C07311=1218.694,48.902,-44.910,-179.073,5.517,148.688
C07312=1218.690,49.151,-44.926,-179.071,5.518,148.687
C07313=1218.684,49.401,-44.942,-179.068,5.518,148.687
C07314=1218.680,49.650,-44.959,-179.065,5.519,148.686
C07315=1218.675,49.900,-44.975,-179.063,5.519,148.685
C07316=1218.670,50.149,-44.991,-179.060,5.520,148.685
C07317=1218.666,50.398,-45.007,-179.058,5.521,148.684
C07318=1218.660,50.648,-45.024,-179.055,5.521,148.684
C07319=1218.655,50.897,-45.041,-179.053,5.522,148.683
C07320=1218.650,51.146,-45.057,-179.050,5.522,148.682
C07321=1218.645,51.396,-45.073,-179.047,5.523,148.682
C07322=1218.641,51.645,-45.090,-179.045,5.524,148.681
C07323=1218.635,51.895,-45.107,-179.043,5.524,148.680
C07324=1218.630,52.145,-45.123,-179.040,5.525,148.680
C07325=1218.625,52.393,-45.139,-179.037,5.526,148.679
C07326=1218.621,52.643,-45.156,-179.035,5.526,148.678
C07327=1218.616,52.892,-45.172,-179.032,5.527,148.678
C07328=1218.611,53.141,-45.189,-179.030,5.528,148.677
C07329=1218.606,53.392,-45.205,-179.027,5.528,148.677
C07330=1218.601,53.641,-45.222,-179.025,5.529,148.676
C07331=1218.596,53.890,-45.238,-179.022,5.529,148.675
C07332=1218.591,54.140,-45.256,-179.019,5.530,148.675
C07333=1218.586,54.388,-45.272,-179.017,5.531,148.674
C07334=1218.581,54.638,-45.289,-179.015,5.531,148.674
C07335=1218.577,54.888,-45.305,-179.012,5.532,148.673
C07336=1218.571,55.156,-45.323,-179.009,5.532,148.672
C07337=1218.566,55.425,-45.341,-179.007,5.533,148.672
C07338=1218.561,55.693,-45.359,-179.004,5.534,148.671
C07339=1218.555,55.962,-45.377,-179.001,5.534,148.670
C07340=1218.550,56.211,-45.393,-178.999,5.535,148.670
C07341=1218.545,56.460,-45.410,-178.996,5.535,148.669
C07342=1218.540,56.710,-45.427,-178.993,5.536,148.668
C07343=1218.535,56.959,-45.443,-178.991,5.538,148.668
C07344=1218.531,57.208,-45.460,-178.988,5.538,148.667
C07345=1218.525,57.458,-45.477,-178.985,5.539,148.666
C07346=1218.520,57.707,-45.493,-178.983,5.539,148.666
C07347=1218.516,57.956,-45.510,-178.980,5.540,148.665
C07348=1218.511,58.206,-45.527,-178.978,5.541,148.665
C07349=1218.506,58.455,-45.544,-178.975,5.541,148.664
C07350=1218.501,58.705,-45.560,-178.973,5.542,148.663
C07351=1218.496,58.954,-45.578,-178.970,5.542,148.663
C07352=1218.491,59.204,-45.594,-178.967,5.543,148.662
C07353=1218.486,59.453,-45.611,-178.965,5.544,148.662
C07354=1218.481,59.702,-45.628,-178.963,5.544,148.661
C07355=1218.477,59.952,-45.644,-178.960,5.545,148.660
C07356=1218.471,60.201,-45.661,-178.957,5.546,148.660
C07357=1218.466,60.450,-45.678,-178.955,5.546,148.659
C07358=1218.462,60.700,-45.695,-178.953,5.547,148.659
C07359=1218.457,60.950,-45.712,-178.950,5.548,148.658
C07360=1218.452,61.199,-45.728,-178.947,5.548,148.657
C07361=1218.447,61.448,-45.746,-178.945,5.549,148.657
C07362=1218.442,61.697,-45.763,-178.943,5.550,148.656
C07363=1218.437,61.947,-45.780,-178.940,5.550,148.655
C07364=1218.432,62.196,-45.797,-178.937,5.551,148.655
C07365=1218.427,62.445,-45.813,-178.935,5.551,148.654
C07366=1218.422,62.695,-45.830,-178.932,5.552,148.653
C07367=1218.418,62.945,-45.847,-178.930,5.553,148.653
C07368=1218.412,63.194,-45.864,-178.927,5.553,148.652
C07369=1218.408,63.442,-45.881,-178.924,5.555,148.652
C07370=1218.402,63.692,-45.899,-178.921,5.555,148.651
C07371=1218.398,63.942,-45.915,-178.919,5.556,148.650
C07372=1218.393,64.192,-45.933,-178.917,5.557,148.650
C07373=1218.388,64.440,-45.949,-178.914,5.557,148.649
C07374=1218.383,64.690,-45.967,-178.911,5.558,148.649
C07375=1218.378,64.939,-45.984,-178.909,5.559,148.648
C07376=1218.373,65.189,-46.001,-178.907,5.560,148.647
C07377=1218.369,65.438,-46.017,-178.904,5.560,148.647
C07378=1218.363,65.687,-46.034,-178.901,5.561,148.646
C07379=1218.359,65.936,-46.052,-178.899,5.561,148.646
C07380=1218.353,66.186,-46.069,-178.897,5.562,148.645
C07381=1218.349,66.436,-46.086,-178.894,5.563,148.644
C07382=1218.344,66.685,-46.104,-178.891,5.563,148.644
C07383=1218.339,66.934,-46.121,-178.889,5.564,148.643
C07384=1218.334,67.183,-46.137,-178.886,5.565,148.642
C07385=1218.328,67.433,-46.155,-178.883,5.566,148.642
C07386=1218.324,67.682,-46.172,-178.881,5.567,148.641
C07387=1218.319,67.932,-46.189,-178.878,5.567,148.641
C07388=1218.315,68.181,-46.206,-178.876,5.568,148.640
C07389=1218.310,68.430,-46.224,-178.873,5.569,148.640
C07390=1218.304,68.680,-46.241,-178.871,5.569,148.639
C07391=1218.299,68.929,-46.257,-178.868,5.570,148.638
C07392=1218.295,69.178,-46.275,-178.866,5.571,148.638
C07393=1218.290,69.428,-46.292,-178.863,5.572,148.637
C07394=1218.285,69.677,-46.310,-178.861,5.572,148.637
C07395=1218.280,69.927,-46.327,-178.858,5.573,148.636
C07396=1218.275,70.176,-46.344,-178.855,5.574,148.635
C07397=1218.271,70.425,-46.362,-178.853,5.575,148.635
C07398=1218.265,70.675,-46.379,-178.850,5.576,148.634
C07399=1218.261,70.923,-46.396,-178.848,5.576,148.633
C07400=1218.255,71.173,-46.413,-178.845,5.577,148.633
C07401=1218.250,71.423,-46.431,-178.843,5.578,148.632
C07402=1218.246,71.672,-46.448,-178.840,5.578,148.632
C07403=1218.241,71.921,-46.465,-178.837,5.579,148.631
C07404=1218.236,72.171,-46.483,-178.835,5.579,148.630
C07405=1218.231,72.420,-46.500,-178.833,5.580,148.630
C07406=1218.226,72.669,-46.518,-178.830,5.581,148.629
C07407=1218.221,72.919,-46.535,-178.827,5.582,148.629
C07408=1218.217,73.168,-46.553,-178.824,5.583,148.628
C07409=1218.212,73.418,-46.570,-178.822,5.584,148.628
C07410=1218.207,73.667,-46.588,-178.820,5.584,148.627
C07411=1218.202,73.917,-46.605,-178.817,5.585,148.626
C07412=1218.197,74.165,-46.622,-178.814,5.585,148.626
C07413=1218.192,74.415,-46.639,-178.812,5.586,148.625
C07414=1218.187,74.664,-46.657,-178.809,5.587,148.624
C07415=1218.182,74.913,-46.675,-178.807,5.588,148.624
C07416=1218.177,75.163,-46.692,-178.804,5.589,148.623
C07417=1218.172,75.412,-46.710,-178.802,5.590,148.623
C07418=1218.167,75.661,-46.727,-178.799,5.590,148.622
C07419=1218.162,75.911,-46.745,-178.796,5.591,148.621
C07420=1218.158,76.160,-46.763,-178.794,5.592,148.621
C07421=1218.153,76.409,-46.780,-178.792,5.593,148.620
C07422=1218.148,76.658,-46.798,-178.789,5.593,148.620
C07423=1218.143,76.908,-46.815,-178.786,5.594,148.619
C07424=1218.138,77.157,-46.833,-178.784,5.595,148.619
C07425=1218.134,77.406,-46.851,-178.781,5.596,148.618
C07426=1218.128,77.656,-46.868,-178.778,5.597,148.617
C07427=1218.124,77.905,-46.886,-178.776,5.598,148.617
C07428=1218.119,78.154,-46.904,-178.774,5.598,148.616
C07429=1218.113,78.404,-46.921,-178.771,5.599,148.616
C07430=1218.109,78.653,-46.939,-178.768,5.599,148.615
C07431=1218.104,78.902,-46.956,-178.766,5.600,148.614
C07432=1218.099,79.151,-46.974,-178.763,5.602,148.614
C07433=1218.094,79.401,-46.992,-178.760,5.602,148.613
C07434=1218.089,79.650,-47.010,-178.758,5.603,148.613
C07435=1218.084,79.900,-47.028,-178.756,5.604,148.612
C07436=1218.079,80.149,-47.046,-178.753,5.604,148.611
C07437=1218.074,80.399,-47.063,-178.750,5.605,148.611
C07438=1218.069,80.648,-47.081,-178.748,5.606,148.610
C07439=1218.066,80.897,-47.099,-178.745,5.607,148.610
C07440=1218.060,81.165,-47.118,-178.742,5.608,148.609
C07441=1218.055,81.434,-47.136,-178.740,5.608,148.608
C07442=1218.050,81.702,-47.156,-178.737,5.610,148.608
C07443=1218.045,81.970,-47.175,-178.734,5.610,148.607
C07444=1218.039,82.220,-47.192,-178.732,5.611,148.607
C07445=1218.034,82.469,-47.210,-178.729,5.612,148.606
C07446=1218.029,82.718,-47.228,-178.727,5.613,148.605
C07447=1218.025,82.968,-47.246,-178.724,5.613,148.605
C07448=1218.020,83.217,-47.265,-178.721,5.615,148.604
C07449=1218.015,83.467,-47.283,-178.719,5.615,148.604
C07450=1218.010,83.716,-47.301,-178.716,5.616,148.603
C07451=1218.005,83.966,-47.318,-178.714,5.617,148.603
C07452=1218.000,84.215,-47.336,-178.711,5.618,148.602
C07453=1217.995,84.464,-47.354,-178.709,5.618,148.601
C07454=1217.990,84.713,-47.372,-178.706,5.620,148.601
C07455=1217.986,84.962,-47.390,-178.703,5.620,148.600
C07456=1217.981,85.211,-47.408,-178.701,5.621,148.599
C07457=1217.976,85.461,-47.426,-178.698,5.622,148.599
C07458=1217.971,85.711,-47.444,-178.696,5.623,148.598
C07459=1217.967,85.960,-47.462,-178.693,5.623,148.598
C07460=1217.962,86.209,-47.480,-178.691,5.625,148.597
C07461=1217.957,86.458,-47.498,-178.688,5.626,148.597
C07462=1217.952,86.707,-47.516,-178.685,5.626,148.596
C07463=1217.947,86.956,-47.534,-178.683,5.627,148.596
C07464=1217.943,87.206,-47.552,-178.681,5.628,148.595
C07465=1217.938,87.455,-47.570,-178.678,5.628,148.594
C07466=1217.933,87.705,-47.588,-178.675,5.630,148.594
C07467=1217.927,87.954,-47.607,-178.673,5.631,148.593
C07468=1217.922,88.203,-47.625,-178.670,5.631,148.593
C07469=1217.917,88.452,-47.643,-178.667,5.632,148.592
C07470=1217.913,88.702,-47.661,-178.665,5.633,148.591
C07471=1217.908,88.952,-47.679,-178.662,5.634,148.591
C07472=1217.903,89.201,-47.697,-178.659,5.635,148.590
C07473=1217.898,89.450,-47.715,-178.657,5.636,148.590
C07474=1217.893,89.699,-47.733,-178.655,5.636,148.589
C07475=1217.889,89.949,-47.751,-178.652,5.637,148.588
C07476=1217.884,90.198,-47.770,-178.649,5.639,148.588
C07477=1217.879,90.447,-47.789,-178.647,5.639,148.587
C07478=1217.874,90.696,-47.807,-178.644,5.640,148.587
C07479=1217.869,90.945,-47.825,-178.642,5.641,148.586
C07480=1217.865,91.195,-47.843,-178.639,5.641,148.586
C07481=1217.860,91.444,-47.861,-178.636,5.643,148.585
C07482=1217.855,91.694,-47.879,-178.634,5.644,148.585
C07483=1217.849,91.942,-47.898,-178.631,5.644,148.584
C07484=1217.845,92.192,-47.916,-178.629,5.645,148.584
C07485=1217.840,92.441,-47.935,-178.627,5.646,148.583
C07486=1217.835,92.691,-47.953,-178.623,5.647,148.582
C07487=1217.830,92.940,-47.971,-178.621,5.648,148.582
C07488=1217.826,93.188,-47.989,-178.619,5.649,148.581
C07489=1217.821,93.439,-48.008,-178.616,5.649,148.581
C07490=1217.816,93.688,-48.026,-178.614,5.650,148.580
C07491=1217.811,93.937,-48.044,-178.611,5.652,148.579
C07492=1217.807,94.186,-48.063,-178.608,5.652,148.579
C07493=1217.801,94.436,-48.082,-178.606,5.653,148.578
C07494=1217.796,94.685,-48.100,-178.603,5.654,148.578
C07495=1217.791,94.934,-48.118,-178.600,5.655,148.577
C07496=1217.787,95.183,-48.137,-178.598,5.656,148.577
C07497=1217.782,95.433,-48.155,-178.595,5.657,148.576
C07498=1217.777,95.682,-48.173,-178.593,5.657,148.575
C07499=1217.772,95.931,-48.192,-178.591,5.658,148.575
C07500=1217.768,96.180,-48.210,-178.588,5.660,148.574
C07501=1217.762,96.430,-48.229,-178.585,5.661,148.574
C07502=1217.758,96.678,-48.248,-178.583,5.661,148.573
C07503=1217.753,96.928,-48.266,-178.580,5.662,148.573
C07504=1217.748,97.178,-48.285,-178.577,5.664,148.572
C07505=1217.743,97.426,-48.303,-178.575,5.664,148.572
C07506=1217.739,97.676,-48.322,-178.572,5.665,148.571
C07507=1217.733,97.926,-48.340,-178.570,5.666,148.570
C07508=1217.729,98.174,-48.359,-178.567,5.667,148.570
C07509=1217.724,98.424,-48.377,-178.564,5.668,148.569
C07510=1217.719,98.673,-48.397,-178.562,5.669,148.569
C07511=1217.714,98.922,-48.415,-178.560,5.669,148.568
C07512=1217.710,99.171,-48.434,-178.557,5.671,148.568
C07513=1217.704,99.421,-48.452,-178.554,5.672,148.567
C07514=1217.699,99.670,-48.470,-178.552,5.672,148.566
C07515=1217.695,99.919,-48.489,-178.549,5.673,148.566
C07516=1217.690,100.169,-48.508,-178.546,5.675,148.565
C07517=1217.685,100.417,-48.527,-178.544,5.676,148.565
C07518=1217.680,100.668,-48.545,-178.542,5.676,148.564
C07519=1217.676,100.916,-48.564,-178.539,5.677,148.564
C07520=1217.671,101.166,-48.583,-178.536,5.679,148.563
C07521=1217.666,101.415,-48.602,-178.534,5.679,148.563
C07522=1217.661,101.664,-48.620,-178.531,5.680,148.562
C07523=1217.656,101.914,-48.639,-178.529,5.681,148.562
C07524=1217.652,102.162,-48.658,-178.526,5.682,148.561
C07525=1217.647,102.412,-48.676,-178.524,5.683,148.561
C07526=1217.642,102.661,-48.696,-178.521,5.684,148.560
C07527=1217.637,102.910,-48.714,-178.518,5.684,148.559
C07528=1217.632,103.160,-48.733,-178.516,5.686,148.559
C07529=1217.627,103.409,-48.751,-178.513,5.687,148.558
C07530=1217.623,103.658,-48.771,-178.511,5.688,148.558
C07531=1217.618,103.907,-48.790,-178.508,5.688,148.557
C07532=1217.612,104.156,-48.808,-178.505,5.690,148.556
C07533=1217.608,104.406,-48.827,-178.503,5.691,148.556
C07534=1217.603,104.655,-48.847,-178.500,5.691,148.555
C07535=1217.599,104.904,-48.865,-178.498,5.693,148.555
C07536=1217.593,105.153,-48.884,-178.495,5.694,148.554
C07537=1217.589,105.403,-48.903,-178.492,5.694,148.554
C07538=1217.584,105.652,-48.922,-178.490,5.695,148.553
C07539=1217.580,105.901,-48.941,-178.487,5.697,148.553
C07540=1217.574,106.150,-48.960,-178.485,5.698,148.552
C07541=1217.569,106.399,-48.978,-178.482,5.698,148.552
C07542=1217.565,106.649,-48.998,-178.479,5.700,148.551
C07543=1217.560,106.898,-49.017,-178.477,5.700,148.551
C07544=1217.555,107.167,-49.037,-178.474,5.701,148.550
C07545=1217.549,107.435,-49.058,-178.471,5.703,148.549
C07546=1217.544,107.703,-49.079,-178.469,5.703,148.549
C07547=1217.539,107.972,-49.099,-178.466,5.705,148.548
C07548=1217.535,108.221,-49.118,-178.463,5.706,148.548
C07549=1217.529,108.470,-49.137,-178.461,5.706,148.547
C07550=1217.525,108.719,-49.156,-178.458,5.708,148.547
C07551=1217.520,108.969,-49.175,-178.455,5.708,148.546
C07552=1217.515,109.218,-49.194,-178.453,5.709,148.546
C07553=1217.510,109.467,-49.213,-178.451,5.710,148.545
C07554=1217.506,109.716,-49.233,-178.448,5.712,148.544
C07555=1217.501,109.965,-49.251,-178.445,5.712,148.544
C07556=1217.496,110.215,-49.270,-178.443,5.713,148.543
C07557=1217.491,110.464,-49.290,-178.440,5.715,148.543
C07558=1217.487,110.713,-49.309,-178.438,5.716,148.542
C07559=1217.482,110.963,-49.328,-178.435,5.716,148.542
C07560=1217.476,111.212,-49.348,-178.432,5.718,148.541
C07561=1217.472,111.461,-49.367,-178.430,5.719,148.541
C07562=1217.467,111.710,-49.386,-178.427,5.719,148.540
C07563=1217.462,111.959,-49.406,-178.425,5.721,148.540
C07564=1217.458,112.208,-49.424,-178.422,5.722,148.539
C07565=1217.453,112.458,-49.443,-178.420,5.723,148.539
C07566=1217.447,112.707,-49.463,-178.417,5.724,148.538
C07567=1217.443,112.956,-49.482,-178.414,5.725,148.537
C07568=1217.439,113.206,-49.501,-178.412,5.726,148.537
C07569=1217.433,113.455,-49.521,-178.409,5.727,148.536
C07570=1217.429,113.704,-49.540,-178.407,5.728,148.536
C07571=1217.424,113.953,-49.559,-178.404,5.729,148.535
C07572=1217.419,114.202,-49.579,-178.402,5.730,148.535
C07573=1217.414,114.451,-49.598,-178.399,5.731,148.534
C07574=1217.409,114.701,-49.618,-178.397,5.732,148.534
C07575=1217.405,114.950,-49.637,-178.394,5.733,148.533
C07576=1217.400,115.199,-49.656,-178.391,5.734,148.533
C07577=1217.395,115.449,-49.676,-178.389,5.735,148.532
C07578=1217.390,115.697,-49.695,-178.386,5.736,148.531
C07579=1217.386,115.947,-49.714,-178.384,5.737,148.531
C07580=1217.381,116.196,-49.734,-178.381,5.738,148.530
C07581=1217.376,116.445,-49.754,-178.378,5.740,148.530
C07582=1217.371,116.694,-49.773,-178.376,5.740,148.529
C07583=1217.366,116.944,-49.793,-178.374,5.741,148.529
C07584=1217.361,117.193,-49.812,-178.370,5.743,148.528
C07585=1217.357,117.442,-49.831,-178.368,5.744,148.528
C07586=1217.352,117.691,-49.851,-178.366,5.744,148.527
C07587=1217.347,117.940,-49.870,-178.363,5.746,148.527
C07588=1217.342,118.190,-49.890,-178.360,5.747,148.526
C07589=1217.338,118.439,-49.910,-178.358,5.748,148.526
C07590=1217.332,118.688,-49.930,-178.355,5.749,148.525
C07591=1217.328,118.937,-49.949,-178.353,5.750,148.525
C07592=1217.324,119.186,-49.968,-178.350,5.751,148.524
C07593=1217.318,119.435,-49.988,-178.348,5.753,148.524
C07594=1217.314,119.685,-50.007,-178.345,5.753,148.523
C07595=1217.309,119.934,-50.028,-178.342,5.755,148.523
C07596=1217.304,120.183,-50.047,-178.340,5.756,148.522
C07597=1217.299,120.432,-50.067,-178.338,5.757,148.522
C07598=1217.294,120.682,-50.086,-178.334,5.758,148.521
C07599=1217.289,120.930,-50.106,-178.332,5.759,148.520
C07600=1217.285,121.179,-50.125,-178.330,5.760,148.520
C07601=1217.281,121.429,-50.145,-178.327,5.761,148.519
C07602=1217.275,121.678,-50.164,-178.324,5.762,148.519
C07603=1217.271,121.927,-50.185,-178.321,5.763,148.518
C07604=1217.266,122.176,-50.204,-178.319,5.764,148.518
C07605=1217.261,122.426,-50.224,-178.317,5.765,148.517
C07606=1217.256,122.674,-50.244,-178.314,5.767,148.517
C07607=1217.251,122.924,-50.264,-178.311,5.767,148.516
C07608=1217.247,123.173,-50.283,-178.309,5.768,148.516
C07609=1217.242,123.422,-50.304,-178.306,5.770,148.515
C07610=1217.237,123.671,-50.323,-178.304,5.771,148.515
C07611=1217.232,123.921,-50.343,-178.301,5.772,148.514
C07612=1217.228,124.170,-50.363,-178.299,5.773,148.514
C07613=1217.223,124.419,-50.383,-178.296,5.774,148.513
C07614=1217.218,124.667,-50.403,-178.293,5.776,148.513
C07615=1217.213,124.917,-50.422,-178.291,5.777,148.512
C07616=1217.209,125.167,-50.442,-178.288,5.778,148.512
C07617=1217.204,125.415,-50.462,-178.286,5.779,148.511
C07618=1217.199,125.665,-50.482,-178.283,5.780,148.511
C07619=1217.194,125.913,-50.502,-178.281,5.781,148.510
C07620=1217.190,126.163,-50.522,-178.278,5.782,148.510
C07621=1217.185,126.412,-50.542,-178.275,5.784,148.509
C07622=1217.180,126.661,-50.562,-178.273,5.784,148.509
C07623=1217.176,126.911,-50.581,-178.271,5.785,148.508
C07624=1217.171,127.159,-50.601,-178.267,5.787,148.508
C07625=1217.165,127.409,-50.622,-178.265,5.788,148.507
C07626=1217.161,127.658,-50.642,-178.262,5.789,148.507
C07627=1217.156,127.908,-50.662,-178.260,5.790,148.506
C07628=1217.151,128.157,-50.682,-178.257,5.791,148.506
C07629=1217.146,128.405,-50.702,-178.255,5.793,148.505
C07630=1217.142,128.654,-50.722,-178.252,5.793,148.505
C07631=1217.137,128.903,-50.742,-178.249,5.795,148.504
C07632=1217.133,129.153,-50.762,-178.247,5.796,148.504
C07633=1217.128,129.402,-50.782,-178.245,5.797,148.503
C07634=1217.123,129.652,-50.802,-178.242,5.798,148.503
C07635=1217.118,129.901,-50.823,-178.239,5.799,148.502
C07636=1217.113,130.149,-50.843,-178.237,5.801,148.502
C07637=1217.108,130.398,-50.862,-178.234,5.801,148.501
C07638=1217.104,130.647,-50.883,-178.231,5.803,148.501
C07639=1217.099,130.897,-50.902,-178.229,5.804,148.500
C07640=1217.094,131.146,-50.923,-178.227,5.805,148.500
C07641=1217.090,131.395,-50.944,-178.224,5.806,148.499
C07642=1217.085,131.645,-50.963,-178.221,5.807,148.499
C07643=1217.080,131.893,-50.983,-178.218,5.809,148.498
C07644=1217.075,132.142,-51.004,-178.216,5.810,148.498
C07645=1217.070,132.392,-51.024,-178.213,5.811,148.497
C07646=1217.065,132.641,-51.044,-178.211,5.812,148.497
C07647=1217.061,132.890,-51.065,-178.208,5.814,148.496
C07648=1217.055,133.159,-51.086,-178.206,5.814,148.496
C07649=1217.051,133.427,-51.108,-178.202,5.816,148.495
C07650=1217.046,133.696,-51.130,-178.200,5.817,148.495
C07651=1217.040,133.965,-51.153,-178.197,5.818,148.494
C07652=1217.036,134.214,-51.173,-178.194,5.820,148.494
C07653=1217.031,134.463,-51.193,-178.192,5.821,148.493
C07654=1217.026,134.712,-51.213,-178.190,5.822,148.493
C07655=1217.021,134.961,-51.234,-178.187,5.823,148.492
C07656=1217.017,135.210,-51.254,-178.184,5.824,148.492
C07657=1217.012,135.459,-51.274,-178.181,5.826,148.491
C07658=1217.007,135.709,-51.295,-178.179,5.827,148.491
C07659=1217.002,135.958,-51.315,-178.177,5.828,148.490
C07660=1216.998,136.206,-51.335,-178.174,5.829,148.490
C07661=1216.993,136.455,-51.356,-178.171,5.831,148.489
C07662=1216.988,136.705,-51.377,-178.169,5.831,148.489
C07663=1216.984,136.954,-51.397,-178.166,5.833,148.488
C07664=1216.979,137.203,-51.417,-178.163,5.834,148.488
C07665=1216.974,137.452,-51.438,-178.161,5.836,148.487
C07666=1216.969,137.701,-51.458,-178.159,5.837,148.487
C07667=1216.964,137.951,-51.479,-178.156,5.837,148.486
C07668=1216.960,138.200,-51.499,-178.153,5.839,148.486
C07669=1216.955,138.449,-51.520,-178.151,5.840,148.485
C07670=1216.950,138.698,-51.541,-178.148,5.841,148.485
C07671=1216.946,138.947,-51.561,-178.146,5.842,148.484
C07672=1216.941,139.196,-51.581,-178.143,5.844,148.484
C07673=1216.936,139.445,-51.602,-178.141,5.845,148.483
C07674=1216.932,139.694,-51.623,-178.137,5.846,148.483
C07675=1216.926,139.943,-51.644,-178.135,5.847,148.482
C07676=1216.922,140.192,-51.664,-178.133,5.849,148.482
C07677=1216.917,140.441,-51.685,-178.130,5.850,148.481
C07678=1216.912,140.690,-51.705,-178.127,5.851,148.481
C07679=1216.908,140.939,-51.726,-178.125,5.852,148.480
C07680=1216.903,141.189,-51.747,-178.122,5.854,148.480
C07681=1216.898,141.437,-51.767,-178.120,5.855,148.479
C07682=1216.893,141.687,-51.788,-178.117,5.856,148.479
C07683=1216.889,141.936,-51.809,-178.115,5.857,148.478
C07684=1216.884,142.185,-51.829,-178.112,5.859,148.478
C07685=1216.879,142.434,-51.850,-178.109,5.860,148.477
C07686=1216.875,142.684,-51.871,-178.107,5.862,148.477
C07687=1216.870,142.933,-51.892,-178.104,5.862,148.476
C07688=1216.865,143.182,-51.913,-178.102,5.864,148.476
C07689=1216.861,143.431,-51.933,-178.099,5.865,148.475
C07690=1216.856,143.680,-51.955,-178.096,5.866,148.475
C07691=1216.851,143.929,-51.975,-178.094,5.867,148.475
C07692=1216.846,144.178,-51.996,-178.091,5.869,148.474
C07693=1216.842,144.427,-52.016,-178.089,5.870,148.474
C07694=1216.836,144.676,-52.037,-178.086,5.872,148.473
C07695=1216.832,144.925,-52.058,-178.084,5.872,148.473
C07696=1216.828,145.174,-52.080,-178.081,5.874,148.472
C07697=1216.823,145.423,-52.100,-178.078,5.875,148.472
C07698=1216.818,145.673,-52.121,-178.076,5.876,148.471
C07699=1216.813,145.922,-52.142,-178.074,5.877,148.471
C07700=1216.808,146.171,-52.162,-178.070,5.879,148.470
C07701=1216.804,146.419,-52.184,-178.068,5.880,148.470
C07702=1216.799,146.668,-52.204,-178.066,5.882,148.470
C07703=1216.794,146.918,-52.225,-178.062,5.883,148.469
C07704=1216.789,147.168,-52.247,-178.060,5.884,148.469
C07705=1216.785,147.416,-52.268,-178.058,5.886,148.468
C07706=1216.780,147.665,-52.289,-178.055,5.887,148.468
C07707=1216.776,147.914,-52.309,-178.052,5.888,148.467
C07708=1216.771,148.163,-52.331,-178.050,5.889,148.467
C07709=1216.766,148.412,-52.352,-178.047,5.891,148.466
C07710=1216.762,148.662,-52.373,-178.045,5.892,148.466
C07711=1216.757,148.910,-52.394,-178.042,5.893,148.465
C07712=1216.752,149.160,-52.415,-178.040,5.894,148.465
C07713=1216.747,149.409,-52.436,-178.037,5.896,148.464
C07714=1216.742,149.657,-52.457,-178.035,5.897,148.464
C07715=1216.737,149.906,-52.478,-178.032,5.898,148.463
C07716=1216.733,150.156,-52.499,-178.029,5.900,148.463
C07717=1216.729,150.405,-52.521,-178.027,5.901,148.462
C07718=1216.723,150.654,-52.542,-178.024,5.903,148.462
C07719=1216.719,150.902,-52.563,-178.022,5.904,148.462
C07720=1216.714,151.152,-52.584,-178.019,5.905,148.461
C07721=1216.710,151.402,-52.605,-178.017,5.906,148.461
C07722=1216.705,151.650,-52.627,-178.014,5.908,148.460
C07723=1216.700,151.899,-52.647,-178.011,5.909,148.460
C07724=1216.695,152.148,-52.669,-178.009,5.910,148.459
C07725=1216.691,152.398,-52.690,-178.006,5.912,148.459
C07726=1216.686,152.646,-52.712,-178.003,5.913,148.458
C07727=1216.681,152.895,-52.732,-178.001,5.915,148.458
C07728=1216.677,153.144,-52.754,-177.999,5.916,148.457
C07729=1216.671,153.393,-52.775,-177.995,5.917,148.457
C07730=1216.667,153.643,-52.797,-177.993,5.918,148.456
C07731=1216.662,153.892,-52.818,-177.991,5.920,148.456
C07732=1216.658,154.140,-52.839,-177.987,5.921,148.456
C07733=1216.653,154.390,-52.860,-177.985,5.922,148.455
C07734=1216.648,154.639,-52.882,-177.983,5.924,148.455
C07735=1216.644,154.887,-52.904,-177.980,5.925,148.454
C07736=1216.638,155.137,-52.925,-177.977,5.927,148.454
C07737=1216.635,155.386,-52.946,-177.975,5.928,148.453
C07738=1216.630,155.635,-52.967,-177.972,5.929,148.453
C07739=1216.625,155.884,-52.989,-177.970,5.931,148.452
C07740=1216.621,156.133,-53.011,-177.967,5.932,148.452
C07741=1216.615,156.382,-53.032,-177.965,5.934,148.452
C07742=1216.610,156.631,-53.053,-177.962,5.934,148.451
C07743=1216.605,156.880,-53.074,-177.959,5.936,148.451
C07744=1216.602,157.129,-53.096,-177.957,5.938,148.450
C07745=1216.597,157.378,-53.117,-177.954,5.939,148.450
C07746=1216.592,157.627,-53.138,-177.952,5.940,148.449
C07747=1216.587,157.876,-53.160,-177.949,5.941,148.449
C07748=1216.583,158.125,-53.182,-177.946,5.943,148.448
C07749=1216.578,158.374,-53.204,-177.944,5.944,148.448
C07750=1216.573,158.624,-53.225,-177.942,5.946,148.448
C07751=1216.568,158.872,-53.247,-177.939,5.947,148.447
C07752=1216.564,159.141,-53.270,-177.936,5.949,148.447
C07753=1216.558,159.410,-53.294,-177.934,5.950,148.446
C07754=1216.553,159.679,-53.317,-177.930,5.951,148.446
C07755=1216.548,159.948,-53.340,-177.928,5.953,148.445
C07756=1216.543,160.197,-53.361,-177.925,5.955,148.445
C07757=1216.539,160.446,-53.384,-177.923,5.956,148.444
C07758=1216.534,160.695,-53.405,-177.920,5.957,148.444
C07759=1216.530,160.944,-53.427,-177.918,5.958,148.443
C07760=1216.525,161.194,-53.448,-177.915,5.960,148.443
C07761=1216.520,161.442,-53.470,-177.912,5.962,148.443
C07762=1216.516,161.692,-53.492,-177.910,5.963,148.442
C07763=1216.511,161.940,-53.514,-177.907,5.964,148.442
C07764=1216.506,162.190,-53.536,-177.904,5.966,148.441
C07765=1216.502,162.438,-53.557,-177.902,5.967,148.441
C07766=1216.497,162.687,-53.579,-177.899,5.969,148.440
C07767=1216.492,162.937,-53.600,-177.897,5.969,148.440
C07768=1216.487,163.185,-53.622,-177.894,5.971,148.439
C07769=1216.483,163.435,-53.644,-177.891,5.973,148.439
C07770=1216.478,163.683,-53.666,-177.889,5.974,148.439
C07771=1216.474,163.933,-53.688,-177.886,5.976,148.438
C07772=1216.469,164.181,-53.710,-177.883,5.977,148.438
C07773=1216.464,164.430,-53.731,-177.881,5.978,148.437
C07774=1216.459,164.680,-53.754,-177.879,5.980,148.437
C07775=1216.454,164.928,-53.776,-177.876,5.982,148.436
C07776=1216.450,165.178,-53.798,-177.873,5.983,148.436
C07777=1216.445,165.426,-53.819,-177.871,5.984,148.436
C07778=1216.441,165.676,-53.841,-177.869,5.985,148.435
C07779=1216.436,165.924,-53.863,-177.866,5.987,148.435
C07780=1216.432,166.174,-53.885,-177.863,5.989,148.434
C07781=1216.427,166.422,-53.907,-177.861,5.990,148.434
C07782=1216.423,166.672,-53.929,-177.858,5.991,148.433
C07783=1216.417,166.921,-53.951,-177.855,5.993,148.433
C07784=1216.413,167.170,-53.973,-177.853,5.994,148.433
C07785=1216.408,167.419,-53.995,-177.850,5.996,148.432
C07786=1216.404,167.668,-54.017,-177.848,5.998,148.432
C07787=1216.399,167.916,-54.039,-177.845,5.998,148.431
C07788=1216.395,168.165,-54.061,-177.842,6.000,148.431
C07789=1216.389,168.414,-54.084,-177.840,6.002,148.430
C07790=1216.385,168.664,-54.106,-177.838,6.003,148.430
C07791=1216.380,168.912,-54.127,-177.834,6.004,148.429
C07792=1216.376,169.162,-54.149,-177.832,6.006,148.429
C07793=1216.371,169.410,-54.171,-177.830,6.007,148.429
C07794=1216.366,169.659,-54.194,-177.827,6.009,148.428
C07795=1216.361,169.908,-54.216,-177.824,6.011,148.428
C07796=1216.357,170.157,-54.238,-177.822,6.011,148.427
C07797=1216.352,170.406,-54.260,-177.819,6.013,148.427
C07798=1216.347,170.656,-54.282,-177.816,6.015,148.427
C07799=1216.343,170.904,-54.305,-177.814,6.016,148.426
C07800=1216.338,171.153,-54.327,-177.811,6.018,148.426
C07801=1216.333,171.402,-54.349,-177.809,6.019,148.425
C07802=1216.328,171.651,-54.371,-177.806,6.020,148.425
C07803=1216.324,171.900,-54.394,-177.804,6.022,148.425
C07804=1216.320,172.149,-54.416,-177.801,6.024,148.424
C07805=1216.315,172.398,-54.438,-177.798,6.025,148.424
C07806=1216.310,172.647,-54.460,-177.796,6.026,148.423
C07807=1216.306,172.896,-54.483,-177.793,6.028,148.423
C07808=1216.301,173.145,-54.505,-177.791,6.030,148.423
C07809=1216.296,173.394,-54.527,-177.788,6.031,148.422
C07810=1216.292,173.643,-54.550,-177.785,6.033,148.422
C07811=1216.286,173.892,-54.572,-177.783,6.034,148.421
C07812=1216.282,174.141,-54.594,-177.781,6.035,148.421
C07813=1216.278,174.390,-54.617,-177.778,6.037,148.420
C07814=1216.272,174.639,-54.639,-177.775,6.039,148.420
C07815=1216.268,174.887,-54.662,-177.773,6.040,148.419
C07816=1216.264,175.136,-54.684,-177.770,6.042,148.419
C07817=1216.259,175.386,-54.706,-177.767,6.043,148.419
C07818=1216.255,175.634,-54.729,-177.765,6.045,148.418
C07819=1216.249,175.883,-54.751,-177.763,6.046,148.418
C07820=1216.245,176.132,-54.774,-177.760,6.048,148.418
C07821=1216.241,176.381,-54.796,-177.757,6.049,148.417
C07822=1216.236,176.630,-54.819,-177.755,6.050,148.417
C07823=1216.231,176.879,-54.841,-177.752,6.052,148.416
C07824=1216.226,177.129,-54.864,-177.749,6.054,148.416
C07825=1216.222,177.377,-54.886,-177.747,6.056,148.416
C07826=1216.217,177.626,-54.909,-177.744,6.057,148.415
C07827=1216.213,177.875,-54.932,-177.741,6.058,148.415
C07828=1216.208,178.123,-54.954,-177.739,6.060,148.414
C07829=1216.203,178.373,-54.977,-177.736,6.062,148.414
C07830=1216.199,178.621,-54.999,-177.734,6.063,148.414
C07831=1216.194,178.870,-55.022,-177.731,6.065,148.413
C07832=1216.190,179.119,-55.044,-177.728,6.066,148.413
C07833=1216.185,179.369,-55.067,-177.726,6.067,148.412
C07834=1216.180,179.617,-55.089,-177.724,6.069,148.412
C07835=1216.175,179.866,-55.112,-177.721,6.071,148.412
C07836=1216.171,180.115,-55.135,-177.718,6.073,148.411
C07837=1216.166,180.364,-55.158,-177.716,6.074,148.411
C07838=1216.161,180.613,-55.180,-177.713,6.075,148.410
C07839=1216.157,180.862,-55.203,-177.710,6.077,148.410
C07840=1216.152,181.111,-55.227,-177.708,6.079,148.410
C07841=1216.148,181.360,-55.249,-177.706,6.080,148.409
C07842=1216.143,181.609,-55.272,-177.703,6.082,148.409
C07843=1216.139,181.857,-55.294,-177.700,6.084,148.408
C07844=1216.134,182.107,-55.317,-177.698,6.085,148.408
C07845=1216.130,182.356,-55.340,-177.695,6.086,148.407
C07846=1216.124,182.604,-55.363,-177.692,6.088,148.407
C07847=1216.120,182.853,-55.385,-177.690,6.090,148.407
C07848=1216.115,183.102,-55.408,-177.687,6.092,148.406
C07849=1216.111,183.351,-55.432,-177.685,6.093,148.406
C07850=1216.106,183.599,-55.454,-177.682,6.094,148.406
C07851=1216.101,183.849,-55.477,-177.680,6.096,148.405
C07852=1216.096,184.098,-55.500,-177.677,6.098,148.405
C07853=1216.092,184.347,-55.523,-177.674,6.100,148.404
C07854=1216.088,184.596,-55.546,-177.672,6.101,148.404
C07855=1216.083,184.844,-55.569,-177.669,6.102,148.404
C07856=1216.078,185.114,-55.594,-177.666,6.104,148.403
C07857=1216.072,185.383,-55.619,-177.663,6.106,148.403
C07858=1216.068,185.653,-55.643,-177.661,6.108,148.402
C07859=1216.063,185.923,-55.668,-177.658,6.109,148.402
C07860=1216.058,186.172,-55.691,-177.655,6.111,148.402
C07861=1216.054,186.420,-55.714,-177.653,6.113,148.401
C07862=1216.049,186.669,-55.738,-177.651,6.114,148.401
C07863=1216.044,186.919,-55.760,-177.648,6.116,148.400
C07864=1216.040,187.168,-55.784,-177.645,6.117,148.400
C07865=1216.035,187.416,-55.806,-177.642,6.119,148.400
C07866=1216.030,187.665,-55.829,-177.640,6.121,148.399
C07867=1216.026,187.914,-55.853,-177.637,6.122,148.399
C07868=1216.022,188.163,-55.875,-177.635,6.124,148.399
C07869=1216.017,188.412,-55.899,-177.632,6.126,148.398
C07870=1216.012,188.661,-55.922,-177.630,6.127,148.398
C07871=1216.008,188.910,-55.946,-177.627,6.129,148.398
C07872=1216.003,189.158,-55.968,-177.624,6.130,148.397
C07873=1215.998,189.407,-55.991,-177.622,6.132,148.397
C07874=1215.994,189.656,-56.015,-177.619,6.134,148.396
C07875=1215.989,189.905,-56.038,-177.616,6.135,148.396
C07876=1215.984,190.154,-56.061,-177.614,6.137,148.396
C07877=1215.980,190.403,-56.084,-177.612,6.138,148.395
C07878=1215.975,190.652,-56.107,-177.609,6.140,148.395
C07879=1215.971,190.901,-56.131,-177.606,6.142,148.394
C07880=1215.966,191.150,-56.154,-177.604,6.144,148.394
C07881=1215.961,191.399,-56.178,-177.601,6.146,148.394
C07882=1215.956,191.647,-56.201,-177.598,6.146,148.393
C07883=1215.952,191.896,-56.223,-177.596,6.148,148.393
C07884=1215.948,192.144,-56.247,-177.593,6.150,148.392
C07885=1215.943,192.393,-56.271,-177.591,6.152,148.392
C07886=1215.938,192.642,-56.294,-177.588,6.154,148.392
C07887=1215.934,192.892,-56.317,-177.585,6.155,148.391
C07888=1215.929,193.141,-56.341,-177.583,6.156,148.391
C07889=1215.924,193.390,-56.364,-177.580,6.158,148.391
C07890=1215.920,193.639,-56.388,-177.578,6.160,148.390
C07891=1215.915,193.887,-56.412,-177.575,6.162,148.390
C07892=1215.911,194.136,-56.434,-177.573,6.164,148.390
C07893=1215.906,194.385,-56.458,-177.570,6.166,148.389
C07894=1215.902,194.634,-56.481,-177.568,6.167,148.389
C07895=1215.897,194.883,-56.504,-177.565,6.168,148.389
C07896=1215.893,195.131,-56.529,-177.562,6.170,148.388
C07897=1215.888,195.380,-56.552,-177.559,6.172,148.388
C07898=1215.883,195.629,-56.575,-177.557,6.174,148.387
C07899=1215.879,195.878,-56.599,-177.554,6.175,148.387
C07900=1215.874,196.127,-56.623,-177.552,6.176,148.387
C07901=1215.869,196.376,-56.646,-177.549,6.178,148.386
C07902=1215.865,196.625,-56.669,-177.547,6.180,148.386
C07903=1215.860,196.873,-56.693,-177.544,6.182,148.386
C07904=1215.856,197.122,-56.717,-177.541,6.184,148.385
C07905=1215.851,197.371,-56.740,-177.539,6.186,148.385
C07906=1215.847,197.620,-56.764,-177.536,6.187,148.385
C07907=1215.842,197.869,-56.788,-177.534,6.188,148.384
C07908=1215.837,198.118,-56.811,-177.531,6.190,148.384
C07909=1215.833,198.366,-56.835,-177.529,6.192,148.383
C07910=1215.828,198.615,-56.858,-177.526,6.194,148.383
C07911=1215.824,198.864,-56.883,-177.523,6.196,148.383
C07912=1215.819,199.113,-56.906,-177.521,6.198,148.382
C07913=1215.814,199.362,-56.929,-177.518,6.199,148.382
C07914=1215.810,199.610,-56.953,-177.516,6.200,148.382
C07915=1215.804,199.859,-56.977,-177.513,6.202,148.381
C07916=1215.800,200.108,-57.001,-177.511,6.204,148.381
C07917=1215.795,200.357,-57.025,-177.508,6.206,148.381
C07918=1215.791,200.605,-57.049,-177.505,6.208,148.380
C07919=1215.787,200.855,-57.072,-177.502,6.209,148.380
C07920=1215.782,201.103,-57.097,-177.500,6.211,148.379
C07921=1215.778,201.353,-57.120,-177.497,6.213,148.379
C07922=1215.773,201.601,-57.144,-177.495,6.214,148.379
C07923=1215.769,201.850,-57.167,-177.492,6.216,148.378
C07924=1215.764,202.099,-57.192,-177.490,6.218,148.378
C07925=1215.759,202.348,-57.215,-177.487,6.220,148.378
C07926=1215.754,202.596,-57.239,-177.484,6.221,148.377
C07927=1215.750,202.845,-57.263,-177.482,6.223,148.377
C07928=1215.745,203.094,-57.287,-177.479,6.225,148.377
C07929=1215.742,203.343,-57.311,-177.476,6.227,148.376
C07930=1215.736,203.592,-57.335,-177.474,6.229,148.376
C07931=1215.732,203.840,-57.359,-177.472,6.230,148.376
C07932=1215.727,204.089,-57.383,-177.469,6.232,148.375
C07933=1215.723,204.338,-57.407,-177.466,6.233,148.375
C07934=1215.718,204.586,-57.431,-177.464,6.235,148.375
C07935=1215.713,204.836,-57.455,-177.461,6.237,148.374
C07936=1215.709,205.085,-57.479,-177.459,6.239,148.374
C07937=1215.705,205.333,-57.503,-177.456,6.241,148.374
C07938=1215.700,205.582,-57.527,-177.453,6.243,148.373
C07939=1215.696,205.831,-57.551,-177.451,6.244,148.373
C07940=1215.690,206.079,-57.575,-177.448,6.246,148.373
C07941=1215.687,206.328,-57.600,-177.445,6.248,148.372
C07942=1215.682,206.577,-57.623,-177.443,6.249,148.372
C07943=1215.677,206.826,-57.648,-177.441,6.251,148.372
C07944=1215.672,207.075,-57.672,-177.438,6.253,148.371
C07945=1215.668,207.323,-57.696,-177.435,6.255,148.371
C07946=1215.663,207.572,-57.719,-177.433,6.257,148.371
C07947=1215.659,207.821,-57.744,-177.430,6.258,148.370
C07948=1215.654,208.070,-57.769,-177.427,6.260,148.370
C07949=1215.650,208.318,-57.793,-177.425,6.262,148.370
C07950=1215.645,208.567,-57.817,-177.422,6.264,148.369
C07951=1215.641,208.817,-57.841,-177.420,6.266,148.369
C07952=1215.636,209.065,-57.865,-177.417,6.268,148.369
C07953=1215.631,209.314,-57.890,-177.415,6.270,148.368
C07954=1215.627,209.562,-57.914,-177.412,6.272,148.368
C07955=1215.622,209.812,-57.939,-177.410,6.273,148.368
C07956=1215.618,210.060,-57.963,-177.407,6.274,148.367
C07957=1215.614,210.309,-57.987,-177.405,6.276,148.367
C07958=1215.608,210.557,-58.012,-177.402,6.278,148.367
C07959=1215.604,210.807,-58.035,-177.399,6.280,148.366
C07960=1215.599,211.077,-58.062,-177.397,6.282,148.366
C07961=1215.594,211.347,-58.089,-177.393,6.284,148.365
C07962=1215.589,211.618,-58.116,-177.390,6.286,148.365
C07963=1215.584,211.887,-58.142,-177.388,6.288,148.365
C07964=1215.580,212.137,-58.166,-177.385,6.290,148.364
C07965=1215.575,212.386,-58.190,-177.383,6.292,148.364
C07966=1215.570,212.635,-58.215,-177.380,6.293,148.364
C07967=1215.566,212.884,-58.239,-177.377,6.295,148.363
C07968=1215.561,213.132,-58.265,-177.375,6.297,148.363
C07969=1215.557,213.380,-58.289,-177.373,6.299,148.363
C07970=1215.552,213.629,-58.313,-177.370,6.301,148.363
C07971=1215.548,213.878,-58.338,-177.367,6.303,148.362
C07972=1215.543,214.127,-58.362,-177.365,6.305,148.362
C07973=1215.539,214.375,-58.386,-177.362,6.307,148.362
C07974=1215.534,214.625,-58.411,-177.359,6.308,148.361
C07975=1215.530,214.873,-58.436,-177.357,6.310,148.361
C07976=1215.525,215.122,-58.460,-177.354,6.312,148.361
C07977=1215.521,215.371,-58.485,-177.351,6.314,148.360
C07978=1215.516,215.620,-58.509,-177.349,6.316,148.360
C07979=1215.512,215.869,-58.534,-177.346,6.318,148.360
C07980=1215.507,216.117,-58.559,-177.344,6.320,148.359
C07981=1215.503,216.365,-58.583,-177.341,6.321,148.359
C07982=1215.498,216.615,-58.608,-177.339,6.322,148.359
C07983=1215.494,216.863,-58.632,-177.336,6.324,148.358
C07984=1215.489,217.112,-58.657,-177.334,6.326,148.358
C07985=1215.484,217.361,-58.683,-177.331,6.328,148.358
C07986=1215.480,217.609,-58.707,-177.329,6.330,148.358
C07987=1215.475,217.858,-58.732,-177.326,6.332,148.357
C07988=1215.471,218.107,-58.756,-177.323,6.334,148.357
C07989=1215.466,218.356,-58.781,-177.321,6.336,148.357
C07990=1215.462,218.604,-58.806,-177.318,6.338,148.356
C07991=1215.457,218.853,-58.830,-177.316,6.339,148.356
C07992=1215.453,219.102,-58.855,-177.313,6.341,148.356
C07993=1215.448,219.350,-58.881,-177.310,6.343,148.355
C07994=1215.443,219.599,-58.905,-177.308,6.345,148.355
C07995=1215.439,219.848,-58.930,-177.306,6.347,148.355
C07996=1215.434,220.096,-58.955,-177.303,6.349,148.354
C07997=1215.430,220.345,-58.980,-177.300,6.351,148.354
C07998=1215.425,220.594,-59.004,-177.298,6.353,148.354
C07999=1215.421,220.843,-59.030,-177.295,6.354,148.353
C08000=1215.417,221.091,-59.054,-177.292,6.356,148.353
C08001=1215.412,221.341,-59.079,-177.290,6.358,148.353
C08002=1215.407,221.589,-59.105,-177.287,6.360,148.353
C08003=1215.403,221.837,-59.129,-177.284,6.362,148.352
C08004=1215.399,222.086,-59.155,-177.282,6.364,148.352
C08005=1215.393,222.335,-59.179,-177.280,6.366,148.352
C08006=1215.389,222.584,-59.204,-177.277,6.368,148.351
C08007=1215.385,222.832,-59.229,-177.274,6.370,148.351
C08008=1215.380,223.081,-59.254,-177.272,6.371,148.351
C08009=1215.376,223.329,-59.279,-177.269,6.373,148.350
C08010=1215.371,223.579,-59.305,-177.266,6.375,148.350
C08011=1215.367,223.827,-59.329,-177.264,6.377,148.350
C08012=1215.362,224.076,-59.354,-177.262,6.379,148.350
C08013=1215.358,224.324,-59.380,-177.259,6.381,148.349
C08014=1215.353,224.574,-59.405,-177.256,6.383,148.349
C08015=1215.348,224.822,-59.430,-177.254,6.385,148.349
C08016=1215.344,225.071,-59.455,-177.251,6.387,148.348
C08017=1215.340,225.319,-59.480,-177.249,6.388,148.348
C08018=1215.335,225.568,-59.506,-177.246,6.391,148.348
C08019=1215.330,225.816,-59.530,-177.244,6.392,148.348
C08020=1215.326,226.065,-59.556,-177.241,6.395,148.347
C08021=1215.321,226.315,-59.581,-177.238,6.397,148.347
C08022=1215.317,226.563,-59.607,-177.235,6.399,148.347
C08023=1215.313,226.811,-59.632,-177.233,6.401,148.346
C08024=1215.308,227.060,-59.656,-177.231,6.403,148.346
C08025=1215.304,227.309,-59.682,-177.228,6.405,148.346
C08026=1215.299,227.557,-59.708,-177.225,6.407,148.346
C08027=1215.294,227.806,-59.733,-177.223,6.408,148.345
C08028=1215.290,228.054,-59.758,-177.220,6.410,148.345
C08029=1215.285,228.303,-59.784,-177.217,6.412,148.345
C08030=1215.281,228.553,-59.809,-177.215,6.414,148.345
C08031=1215.276,228.801,-59.834,-177.213,6.416,148.344
C08032=1215.272,229.050,-59.860,-177.210,6.418,148.344
C08033=1215.267,229.298,-59.885,-177.207,6.420,148.344
C08034=1215.263,229.547,-59.910,-177.205,6.422,148.343
C08035=1215.259,229.796,-59.935,-177.202,6.424,148.343
C08036=1215.254,230.044,-59.961,-177.200,6.426,148.343
C08037=1215.250,230.293,-59.987,-177.197,6.428,148.342
C08038=1215.245,230.542,-60.012,-177.195,6.430,148.342
C08039=1215.241,230.790,-60.037,-177.192,6.431,148.342
C08040=1215.236,231.039,-60.063,-177.189,6.433,148.342
C08041=1215.231,231.287,-60.088,-177.187,6.435,148.341
C08042=1215.227,231.536,-60.114,-177.185,6.437,148.341
C08043=1215.223,231.785,-60.139,-177.182,6.439,148.341
C08044=1215.218,232.033,-60.164,-177.179,6.441,148.340
C08045=1215.214,232.282,-60.190,-177.177,6.443,148.340
C08046=1215.209,232.531,-60.216,-177.175,6.445,148.340
C08047=1215.204,232.779,-60.242,-177.171,6.448,148.340
C08048=1215.200,233.028,-60.268,-177.169,6.450,148.339
C08049=1215.195,233.277,-60.293,-177.166,6.451,148.339
C08050=1215.191,233.525,-60.319,-177.164,6.454,148.339
C08051=1215.186,233.774,-60.344,-177.161,6.455,148.339
C08052=1215.182,234.023,-60.370,-177.159,6.457,148.338
C08053=1215.177,234.271,-60.396,-177.156,6.459,148.338
C08054=1215.173,234.520,-60.421,-177.154,6.461,148.338
C08055=1215.169,234.768,-60.447,-177.151,6.463,148.338
C08056=1215.164,235.016,-60.472,-177.149,6.465,148.337
C08057=1215.160,235.265,-60.498,-177.146,6.467,148.337
C08058=1215.155,235.514,-60.525,-177.144,6.469,148.337
C08059=1215.151,235.763,-60.550,-177.141,6.471,148.337
C08060=1215.146,236.011,-60.576,-177.139,6.473,148.336
C08061=1215.142,236.260,-60.601,-177.136,6.475,148.336
C08062=1215.137,236.509,-60.627,-177.133,6.477,148.336
C08063=1215.133,236.758,-60.653,-177.131,6.480,148.336
C08064=1215.128,237.029,-60.681,-177.128,6.481,148.335
C08065=1215.123,237.301,-60.709,-177.126,6.483,148.335
C08066=1215.117,237.572,-60.738,-177.122,6.486,148.335
C08067=1215.113,237.844,-60.766,-177.120,6.488,148.334
C08068=1215.109,238.092,-60.791,-177.117,6.490,148.334
C08069=1215.104,238.340,-60.818,-177.114,6.492,148.334
C08070=1215.100,238.589,-60.843,-177.112,6.494,148.334
C08071=1215.095,238.838,-60.870,-177.110,6.496,148.333
C08072=1215.091,239.087,-60.895,-177.107,6.498,148.333
C08073=1215.086,239.335,-60.921,-177.104,6.500,148.333
C08074=1215.082,239.584,-60.946,-177.102,6.502,148.333
C08075=1215.077,239.832,-60.974,-177.099,6.504,148.332
C08076=1215.073,240.081,-60.999,-177.097,6.506,148.332
C08077=1215.068,240.330,-61.025,-177.094,6.508,148.332
C08078=1215.064,240.578,-61.051,-177.092,6.510,148.332
C08079=1215.059,240.826,-61.078,-177.089,6.512,148.331
C08080=1215.055,241.075,-61.103,-177.087,6.514,148.331
C08081=1215.051,241.324,-61.129,-177.084,6.516,148.331
C08082=1215.046,241.573,-61.155,-177.081,6.519,148.331
C08083=1215.042,241.821,-61.182,-177.079,6.521,148.330
C08084=1215.037,242.069,-61.207,-177.076,6.523,148.330
C08085=1215.033,242.318,-61.233,-177.074,6.525,148.330
C08086=1215.028,242.567,-61.260,-177.071,6.526,148.330
C08087=1215.024,242.815,-61.286,-177.069,6.528,148.329
C08088=1215.019,243.064,-61.312,-177.066,6.530,148.329
C08089=1215.015,243.313,-61.339,-177.064,6.532,148.329
C08090=1215.011,243.561,-61.364,-177.061,6.534,148.328
C08091=1215.005,243.809,-61.391,-177.058,6.537,148.328
C08092=1215.001,244.058,-61.417,-177.056,6.539,148.328
C08093=1214.997,244.307,-61.443,-177.053,6.541,148.328
C08094=1214.992,244.555,-61.470,-177.051,6.543,148.328
C08095=1214.988,244.804,-61.495,-177.048,6.545,148.327
C08096=1214.983,245.053,-61.522,-177.046,6.547,148.327
C08097=1214.979,245.301,-61.548,-177.044,6.549,148.327
C08098=1214.975,245.550,-61.575,-177.041,6.551,148.327
C08099=1214.970,245.798,-61.601,-177.038,6.554,148.326
C08100=1214.966,246.046,-61.627,-177.035,6.555,148.326
C08101=1214.961,246.295,-61.653,-177.033,6.558,148.326
C08102=1214.957,246.544,-61.680,-177.031,6.560,148.326
C08103=1214.952,246.793,-61.706,-177.028,6.561,148.325
C08104=1214.948,247.041,-61.733,-177.026,6.564,148.325
C08105=1214.943,247.290,-61.759,-177.023,6.565,148.325
C08106=1214.939,247.538,-61.785,-177.021,6.567,148.325
C08107=1214.934,247.787,-61.812,-177.018,6.570,148.325
C08108=1214.930,248.035,-61.838,-177.015,6.572,148.324
C08109=1214.925,248.285,-61.865,-177.013,6.574,148.324
C08110=1214.921,248.533,-61.891,-177.010,6.576,148.324
C08111=1214.917,248.781,-61.918,-177.008,6.578,148.324
C08112=1214.912,249.030,-61.944,-177.006,6.580,148.323
C08113=1214.908,249.279,-61.971,-177.003,6.583,148.323
C08114=1214.904,249.527,-61.997,-177.000,6.585,148.323
C08115=1214.899,249.776,-62.024,-176.998,6.587,148.323
C08116=1214.894,250.023,-62.050,-176.995,6.589,148.322
C08117=1214.890,250.272,-62.077,-176.993,6.591,148.322
C08118=1214.885,250.521,-62.103,-176.990,6.593,148.322
C08119=1214.881,250.769,-62.130,-176.988,6.595,148.322
C08120=1214.876,251.018,-62.157,-176.985,6.598,148.322
C08121=1214.872,251.266,-62.183,-176.982,6.600,148.321
C08122=1214.867,251.515,-62.210,-176.980,6.602,148.321
C08123=1214.863,251.763,-62.237,-176.977,6.603,148.321
C08124=1214.859,252.012,-62.263,-176.975,6.606,148.321
C08125=1214.855,252.261,-62.291,-176.972,6.608,148.320
C08126=1214.850,252.510,-62.316,-176.970,6.610,148.320
C08127=1214.846,252.758,-62.343,-176.967,6.612,148.320
C08128=1214.841,253.007,-62.370,-176.965,6.614,148.320
C08129=1214.837,253.255,-62.397,-176.962,6.616,148.320
C08130=1214.833,253.503,-62.424,-176.960,6.618,148.319
C08131=1214.828,253.752,-62.450,-176.957,6.621,148.319
C08132=1214.824,254.001,-62.477,-176.954,6.623,148.319
C08133=1214.819,254.249,-62.504,-176.952,6.625,148.319
C08134=1214.814,254.498,-62.531,-176.950,6.627,148.319
C08135=1214.810,254.746,-62.558,-176.947,6.629,148.318
C08136=1214.806,254.994,-62.584,-176.944,6.632,148.318
C08137=1214.801,255.243,-62.612,-176.942,6.634,148.318
C08138=1214.796,255.491,-62.639,-176.939,6.636,148.318
C08139=1214.793,255.739,-62.665,-176.937,6.638,148.318
C08140=1214.788,255.988,-62.692,-176.934,6.640,148.317
C08141=1214.783,256.236,-62.719,-176.932,6.643,148.317
C08142=1214.779,256.486,-62.746,-176.929,6.645,148.317
C08143=1214.775,256.734,-62.772,-176.927,6.647,148.317
C08144=1214.770,256.983,-62.799,-176.924,6.649,148.317
C08145=1214.766,257.231,-62.826,-176.922,6.651,148.316
C08146=1214.761,257.480,-62.854,-176.919,6.654,148.316
C08147=1214.757,257.728,-62.881,-176.916,6.656,148.316
C08148=1214.753,257.976,-62.908,-176.914,6.658,148.316
C08149=1214.748,258.224,-62.935,-176.912,6.660,148.315
C08150=1214.743,258.473,-62.962,-176.909,6.662,148.315
C08151=1214.739,258.722,-62.989,-176.906,6.665,148.315
C08152=1214.735,258.971,-63.016,-176.904,6.666,148.315
C08153=1214.730,259.219,-63.043,-176.902,6.669,148.315
C08154=1214.726,259.467,-63.070,-176.899,6.671,148.314
C08155=1214.721,259.716,-63.097,-176.897,6.673,148.314
C08156=1214.717,259.964,-63.124,-176.894,6.675,148.314
C08157=1214.713,260.214,-63.151,-176.891,6.677,148.314
C08158=1214.708,260.461,-63.179,-176.889,6.679,148.314
C08159=1214.704,260.710,-63.206,-176.886,6.681,148.313
C08160=1214.699,260.958,-63.233,-176.884,6.684,148.313
C08161=1214.694,261.207,-63.260,-176.881,6.686,148.313
C08162=1214.691,261.455,-63.287,-176.879,6.688,148.313
C08163=1214.687,261.704,-63.315,-176.876,6.690,148.313
C08164=1214.682,261.952,-63.342,-176.874,6.693,148.313
C08165=1214.677,262.201,-63.369,-176.871,6.695,148.312
C08166=1214.673,262.449,-63.396,-176.869,6.697,148.312
C08167=1214.668,262.698,-63.423,-176.866,6.699,148.312
C08168=1214.663,262.971,-63.454,-176.863,6.702,148.312
C08169=1214.659,263.243,-63.484,-176.861,6.704,148.312
C08170=1214.654,263.516,-63.514,-176.858,6.707,148.311
C08171=1214.649,263.788,-63.544,-176.855,6.710,148.311
C08172=1214.644,264.037,-63.571,-176.852,6.712,148.311
C08173=1214.641,264.285,-63.599,-176.850,6.714,148.311
C08174=1214.636,264.534,-63.626,-176.848,6.716,148.311
C08175=1214.631,264.782,-63.653,-176.845,6.719,148.310
C08176=1214.627,265.030,-63.681,-176.842,6.721,148.310
C08177=1214.623,265.279,-63.708,-176.840,6.723,148.310
C08178=1214.618,265.528,-63.735,-176.838,6.725,148.310
C08179=1214.614,265.776,-63.763,-176.835,6.728,148.310
C08180=1214.610,266.025,-63.791,-176.832,6.730,148.310
C08181=1214.606,266.273,-63.818,-176.830,6.732,148.309
C08182=1214.601,266.521,-63.845,-176.828,6.734,148.309
C08183=1214.596,266.769,-63.874,-176.824,6.736,148.309
C08184=1214.592,267.019,-63.901,-176.822,6.739,148.309
C08185=1214.587,267.267,-63.928,-176.820,6.741,148.309
C08186=1214.583,267.515,-63.956,-176.818,6.743,148.308
C08187=1214.579,267.764,-63.983,-176.814,6.745,148.308
C08188=1214.574,268.012,-64.011,-176.812,6.748,148.308
C08189=1214.570,268.261,-64.038,-176.810,6.750,148.308
C08190=1214.565,268.508,-64.066,-176.807,6.753,148.308
C08191=1214.562,268.757,-64.094,-176.804,6.754,148.308
C08192=1214.556,269.006,-64.122,-176.802,6.757,148.307
C08193=1214.552,269.254,-64.150,-176.800,6.759,148.307
C08194=1214.548,269.503,-64.177,-176.797,6.762,148.307
C08195=1214.543,269.751,-64.205,-176.795,6.764,148.307
C08196=1214.539,269.999,-64.232,-176.792,6.766,148.307
C08197=1214.535,270.248,-64.260,-176.790,6.769,148.307
C08198=1214.530,270.496,-64.288,-176.787,6.770,148.306
C08199=1214.526,270.745,-64.316,-176.785,6.773,148.306
C08200=1214.522,270.993,-64.344,-176.782,6.775,148.306
C08201=1214.517,271.241,-64.371,-176.780,6.778,148.306
C08202=1214.513,271.490,-64.399,-176.777,6.779,148.306
C08203=1214.508,271.738,-64.427,-176.775,6.782,148.306
C08204=1214.504,271.986,-64.455,-176.772,6.785,148.306
C08205=1214.500,272.235,-64.482,-176.769,6.787,148.305
C08206=1214.495,272.483,-64.510,-176.767,6.789,148.305
C08207=1214.491,272.732,-64.539,-176.764,6.791,148.305
C08208=1214.486,272.981,-64.566,-176.762,6.794,148.305
C08209=1214.482,273.229,-64.594,-176.759,6.796,148.305
C08210=1214.478,273.477,-64.622,-176.757,6.799,148.305
C08211=1214.473,273.725,-64.650,-176.755,6.801,148.304
C08212=1214.469,273.974,-64.678,-176.752,6.803,148.304
C08213=1214.465,274.222,-64.705,-176.750,6.805,148.304
C08214=1214.460,274.471,-64.734,-176.747,6.808,148.304
C08215=1214.456,274.719,-64.762,-176.745,6.810,148.304
C08216=1214.451,274.967,-64.790,-176.742,6.812,148.304
C08217=1214.447,275.216,-64.818,-176.739,6.815,148.303
C08218=1214.443,275.464,-64.846,-176.737,6.817,148.303
C08219=1214.439,275.713,-64.874,-176.735,6.819,148.303
C08220=1214.433,275.961,-64.902,-176.732,6.822,148.303
C08221=1214.430,276.210,-64.930,-176.730,6.824,148.303
C08222=1214.425,276.458,-64.958,-176.727,6.826,148.303
C08223=1214.421,276.707,-64.987,-176.724,6.829,148.303
C08224=1214.416,276.954,-65.014,-176.722,6.831,148.302
C08225=1214.412,277.203,-65.043,-176.720,6.833,148.302
C08226=1214.408,277.451,-65.071,-176.717,6.836,148.302
C08227=1214.404,277.700,-65.099,-176.714,6.838,148.302
C08228=1214.399,277.948,-65.128,-176.712,6.840,148.302
C08229=1214.395,278.197,-65.156,-176.710,6.843,148.302
C08230=1214.390,278.445,-65.184,-176.707,6.845,148.302
C08231=1214.386,278.693,-65.212,-176.705,6.847,148.302
C08232=1214.382,278.941,-65.240,-176.702,6.850,148.301
C08233=1214.377,279.190,-65.269,-176.700,6.852,148.301
C08234=1214.373,279.438,-65.296,-176.697,6.855,148.301
C08235=1214.369,279.687,-65.325,-176.694,6.857,148.301
C08236=1214.364,279.935,-65.353,-176.692,6.859,148.301
C08237=1214.360,280.184,-65.382,-176.690,6.862,148.301
C08238=1214.355,280.431,-65.409,-176.687,6.864,148.300
C08239=1214.351,280.680,-65.438,-176.685,6.866,148.300
C08240=1214.347,280.928,-65.466,-176.682,6.869,148.300
C08241=1214.342,281.176,-65.495,-176.680,6.871,148.300
C08242=1214.339,281.425,-65.524,-176.677,6.873,148.300
C08243=1214.333,281.673,-65.552,-176.675,6.876,148.300
C08244=1214.330,281.922,-65.580,-176.672,6.878,148.300
C08245=1214.325,282.170,-65.608,-176.670,6.881,148.300
C08246=1214.321,282.419,-65.637,-176.667,6.884,148.300
C08247=1214.316,282.666,-65.666,-176.665,6.885,148.299
C08248=1214.312,282.915,-65.694,-176.662,6.888,148.299
C08249=1214.308,283.164,-65.723,-176.660,6.891,148.299
C08250=1214.303,283.412,-65.751,-176.658,6.893,148.299
C08251=1214.299,283.660,-65.779,-176.655,6.896,148.299
C08252=1214.294,283.908,-65.808,-176.652,6.898,148.299
C08253=1214.290,284.157,-65.837,-176.650,6.900,148.299
C08254=1214.286,284.405,-65.865,-176.647,6.903,148.299
C08255=1214.281,284.653,-65.894,-176.645,6.905,148.298
C08256=1214.277,284.902,-65.922,-176.642,6.908,148.298
C08257=1214.273,285.150,-65.951,-176.640,6.910,148.298
C08258=1214.268,285.399,-65.979,-176.638,6.912,148.298
C08259=1214.264,285.647,-66.008,-176.635,6.915,148.298
C08260=1214.259,285.895,-66.037,-176.633,6.917,148.298
C08261=1214.255,286.143,-66.066,-176.630,6.920,148.298
C08262=1214.251,286.392,-66.094,-176.628,6.922,148.298
C08263=1214.246,286.640,-66.123,-176.625,6.924,148.298
C08264=1214.242,286.888,-66.152,-176.623,6.927,148.298
C08265=1214.238,287.137,-66.181,-176.620,6.929,148.297
C08266=1214.234,287.384,-66.209,-176.617,6.932,148.297
C08267=1214.229,287.633,-66.238,-176.615,6.935,148.297
C08268=1214.225,287.882,-66.267,-176.613,6.937,148.297
C08269=1214.221,288.129,-66.295,-176.610,6.939,148.297
C08270=1214.216,288.378,-66.324,-176.608,6.942,148.297
C08271=1214.212,288.626,-66.353,-176.605,6.945,148.297
C08272=1214.207,288.901,-66.385,-176.603,6.947,148.297
C08273=1214.202,289.175,-66.417,-176.600,6.950,148.297
C08274=1214.198,289.449,-66.449,-176.597,6.953,148.297
C08275=1214.193,289.723,-66.481,-176.594,6.955,148.296
C08276=1214.188,289.971,-66.509,-176.592,6.958,148.296
C08277=1214.184,290.220,-66.539,-176.590,6.960,148.296
C08278=1214.180,290.468,-66.568,-176.587,6.963,148.296
C08279=1214.176,290.717,-66.596,-176.585,6.965,148.296
C08280=1214.171,290.964,-66.625,-176.582,6.968,148.296
C08281=1214.167,291.213,-66.654,-176.580,6.970,148.296
C08282=1214.162,291.461,-66.683,-176.578,6.972,148.296
C08283=1214.158,291.709,-66.713,-176.575,6.975,148.296
C08284=1214.153,291.958,-66.741,-176.573,6.977,148.296
C08285=1214.150,292.206,-66.770,-176.570,6.980,148.295
C08286=1214.146,292.454,-66.800,-176.568,6.982,148.295
C08287=1214.141,292.703,-66.828,-176.565,6.985,148.295
C08288=1214.137,292.951,-66.858,-176.563,6.987,148.295
C08289=1214.132,293.199,-66.887,-176.561,6.990,148.295
C08290=1214.128,293.448,-66.916,-176.558,6.992,148.295
C08291=1214.123,293.696,-66.945,-176.555,6.995,148.295
C08292=1214.119,293.944,-66.975,-176.553,6.998,148.295
C08293=1214.114,294.192,-67.004,-176.551,7.000,148.295
C08294=1214.111,294.440,-67.032,-176.548,7.003,148.295
C08295=1214.106,294.688,-67.061,-176.546,7.005,148.295
C08296=1214.102,294.937,-67.091,-176.543,7.007,148.294
C08297=1214.098,295.185,-67.120,-176.541,7.010,148.294
C08298=1214.094,295.434,-67.149,-176.538,7.012,148.294
C08299=1214.089,295.681,-67.178,-176.536,7.015,148.294
C08300=1214.085,295.930,-67.207,-176.534,7.017,148.294
C08301=1214.080,296.178,-67.237,-176.531,7.020,148.294
C08302=1214.076,296.426,-67.266,-176.529,7.023,148.294
C08303=1214.072,296.675,-67.296,-176.526,7.025,148.294
C08304=1214.068,296.923,-67.325,-176.524,7.028,148.294
C08305=1214.063,297.172,-67.354,-176.521,7.030,148.294
C08306=1214.059,297.419,-67.383,-176.519,7.033,148.294
C08307=1214.054,297.668,-67.412,-176.517,7.035,148.294
C08308=1214.050,297.916,-67.442,-176.514,7.038,148.294
C08309=1214.046,298.164,-67.471,-176.512,7.040,148.294
C08310=1214.042,298.412,-67.501,-176.509,7.043,148.294
C08311=1214.038,298.661,-67.530,-176.507,7.046,148.294
C08312=1214.034,298.909,-67.560,-176.504,7.049,148.294
C08313=1214.029,299.157,-67.589,-176.502,7.050,148.293
C08314=1214.024,299.405,-67.619,-176.499,7.054,148.293
C08315=1214.020,299.653,-67.648,-176.497,7.056,148.293
C08316=1214.016,299.902,-67.678,-176.495,7.058,148.293
C08317=1214.011,300.150,-67.707,-176.492,7.061,148.293
C08318=1214.007,300.398,-67.737,-176.490,7.063,148.293
C08319=1214.003,300.646,-67.766,-176.487,7.066,148.293
C08320=1213.999,300.895,-67.796,-176.485,7.068,148.293
C08321=1213.995,301.143,-67.825,-176.483,7.071,148.293
C08322=1213.990,301.391,-67.855,-176.480,7.074,148.293
C08323=1213.986,301.639,-67.885,-176.478,7.077,148.293
C08324=1213.982,301.887,-67.915,-176.476,7.079,148.293
C08325=1213.977,302.136,-67.944,-176.473,7.082,148.293
C08326=1213.973,302.384,-67.974,-176.471,7.084,148.293
C08327=1213.969,302.632,-68.003,-176.468,7.087,148.293
C08328=1213.964,302.880,-68.033,-176.466,7.089,148.293
C08329=1213.959,303.128,-68.062,-176.463,7.092,148.293
C08330=1213.956,303.376,-68.092,-176.461,7.095,148.293
C08331=1213.951,303.624,-68.122,-176.458,7.097,148.292
C08332=1213.947,303.872,-68.151,-176.456,7.100,148.292
C08333=1213.942,304.121,-68.181,-176.454,7.102,148.292
C08334=1213.938,304.369,-68.211,-176.451,7.105,148.292
C08335=1213.934,304.617,-68.241,-176.449,7.107,148.292
C08336=1213.930,304.865,-68.270,-176.446,7.110,148.292
C08337=1213.925,305.114,-68.300,-176.444,7.112,148.292
C08338=1213.921,305.361,-68.331,-176.442,7.115,148.292
C08339=1213.917,305.610,-68.360,-176.440,7.118,148.292
C08340=1213.912,305.858,-68.390,-176.437,7.121,148.292
C08341=1213.908,306.107,-68.420,-176.435,7.123,148.292
C08342=1213.904,306.354,-68.450,-176.433,7.126,148.292
C08343=1213.900,306.602,-68.479,-176.430,7.128,148.292
C08344=1213.895,306.851,-68.509,-176.428,7.131,148.292
C08345=1213.891,307.099,-68.539,-176.426,7.134,148.292
C08346=1213.887,307.347,-68.569,-176.423,7.137,148.292
C08347=1213.883,307.596,-68.600,-176.421,7.139,148.292
C08348=1213.879,307.844,-68.629,-176.418,7.142,148.292
C08349=1213.875,308.092,-68.659,-176.416,7.144,148.292
C08350=1213.870,308.340,-68.690,-176.413,7.147,148.292
C08351=1213.866,308.588,-68.719,-176.411,7.149,148.292
C08352=1213.861,308.836,-68.750,-176.409,7.152,148.292
C08353=1213.857,309.085,-68.779,-176.406,7.154,148.292
C08354=1213.853,309.332,-68.810,-176.404,7.158,148.292
C08355=1213.848,309.581,-68.840,-176.402,7.160,148.292
C08356=1213.844,309.828,-68.870,-176.399,7.163,148.292
C08357=1213.839,310.077,-68.900,-176.397,7.165,148.292
C08358=1213.835,310.325,-68.930,-176.395,7.168,148.292
C08359=1213.831,310.573,-68.959,-176.393,7.171,148.292
C08360=1213.827,310.822,-68.991,-176.390,7.174,148.292
C08361=1213.823,311.070,-69.020,-176.388,7.176,148.292
C08362=1213.818,311.318,-69.051,-176.385,7.179,148.292
C08363=1213.815,311.566,-69.081,-176.383,7.181,148.292
C08364=1213.810,311.814,-69.111,-176.380,7.184,148.292
C08365=1213.806,312.062,-69.141,-176.378,7.186,148.292
C08366=1213.801,312.310,-69.171,-176.376,7.190,148.292
C08367=1213.797,312.558,-69.201,-176.374,7.192,148.292
C08368=1213.793,312.807,-69.232,-176.371,7.195,148.292
C08369=1213.789,313.055,-69.262,-176.369,7.197,148.292
C08370=1213.784,313.303,-69.293,-176.366,7.200,148.292
C08371=1213.780,313.550,-69.323,-176.364,7.202,148.292
C08372=1213.775,313.799,-69.353,-176.362,7.205,148.292
C08373=1213.772,314.047,-69.383,-176.360,7.208,148.292
C08374=1213.768,314.295,-69.414,-176.357,7.211,148.292
C08375=1213.763,314.544,-69.444,-176.355,7.213,148.292
C08376=1213.759,314.819,-69.478,-176.352,7.216,148.292
C08377=1213.754,315.095,-69.512,-176.350,7.219,148.292
C08378=1213.749,315.372,-69.546,-176.347,7.222,148.292
C08379=1213.745,315.647,-69.579,-176.344,7.225,148.292
C08380=1213.740,315.896,-69.610,-176.343,7.228,148.292
C08381=1213.735,316.144,-69.640,-176.340,7.231,148.292
C08382=1213.731,316.391,-69.670,-176.338,7.233,148.292
C08383=1213.727,316.640,-69.702,-176.335,7.236,148.292
C08384=1213.723,316.888,-69.732,-176.333,7.238,148.292
C08385=1213.719,317.136,-69.763,-176.331,7.242,148.292
C08386=1213.714,317.384,-69.793,-176.329,7.244,148.292
C08387=1213.711,317.633,-69.823,-176.326,7.247,148.292
C08388=1213.706,317.880,-69.854,-176.324,7.250,148.292
C08389=1213.701,318.128,-69.885,-176.322,7.252,148.292
C08390=1213.697,318.376,-69.915,-176.319,7.256,148.292
C08391=1213.693,318.625,-69.946,-176.317,7.258,148.292
C08392=1213.689,318.873,-69.977,-176.314,7.261,148.292
C08393=1213.685,319.120,-70.007,-176.313,7.263,148.292
C08394=1213.680,319.368,-70.038,-176.310,7.266,148.292
C08395=1213.676,319.617,-70.069,-176.308,7.269,148.292
C08396=1213.672,319.865,-70.099,-176.306,7.272,148.293
C08397=1213.668,320.113,-70.130,-176.304,7.274,148.293
C08398=1213.663,320.361,-70.160,-176.301,7.277,148.293
C08399=1213.659,320.609,-70.192,-176.299,7.279,148.292
C08400=1213.655,320.857,-70.222,-176.297,7.283,148.293
C08401=1213.651,321.105,-70.253,-176.295,7.285,148.293
C08402=1213.647,321.353,-70.284,-176.292,7.288,148.293
C08403=1213.642,321.601,-70.314,-176.290,7.290,148.293
C08404=1213.638,321.849,-70.345,-176.288,7.294,148.293
C08405=1213.634,322.098,-70.376,-176.286,7.296,148.293
C08406=1213.630,322.346,-70.406,-176.283,7.299,148.293
C08407=1213.625,322.594,-70.437,-176.281,7.301,148.293
C08408=1213.621,322.842,-70.468,-176.279,7.304,148.293
C08409=1213.617,323.089,-70.499,-176.277,7.307,148.293
C08410=1213.613,323.337,-70.530,-176.274,7.310,148.293
C08411=1213.609,323.586,-70.561,-176.273,7.312,148.293
C08412=1213.604,323.834,-70.592,-176.270,7.315,148.293
C08413=1213.600,324.082,-70.623,-176.267,7.318,148.293
C08414=1213.596,324.330,-70.654,-176.266,7.321,148.293
C08415=1213.592,324.578,-70.685,-176.263,7.324,148.293
C08416=1213.587,324.825,-70.715,-176.261,7.326,148.293
C08417=1213.583,325.074,-70.747,-176.259,7.330,148.294
C08418=1213.579,325.322,-70.777,-176.256,7.332,148.294
C08419=1213.575,325.570,-70.809,-176.254,7.335,148.294
C08420=1213.570,325.818,-70.840,-176.252,7.337,148.294
C08421=1213.566,326.066,-70.871,-176.249,7.340,148.294
C08422=1213.562,326.315,-70.902,-176.248,7.343,148.294
C08423=1213.558,326.562,-70.933,-176.245,7.346,148.294
C08424=1213.554,326.810,-70.964,-176.244,7.348,148.294
C08425=1213.550,327.058,-70.995,-176.241,7.352,148.294
C08426=1213.545,327.306,-71.026,-176.239,7.354,148.294
C08427=1213.541,327.554,-71.057,-176.237,7.357,148.294
C08428=1213.537,327.802,-71.088,-176.235,7.360,148.294
C08429=1213.533,328.050,-71.120,-176.232,7.363,148.294
C08430=1213.528,328.298,-71.151,-176.231,7.365,148.295
C08431=1213.525,328.546,-71.182,-176.228,7.368,148.295
C08432=1213.520,328.794,-71.213,-176.226,7.371,148.295
C08433=1213.515,329.042,-71.244,-176.224,7.374,148.295
C08434=1213.512,329.290,-71.276,-176.221,7.377,148.295
C08435=1213.507,329.538,-71.307,-176.219,7.379,148.295
C08436=1213.503,329.786,-71.338,-176.217,7.383,148.295
C08437=1213.499,330.034,-71.369,-176.215,7.385,148.295
C08438=1213.495,330.282,-71.401,-176.213,7.388,148.295
C08439=1213.490,330.530,-71.432,-176.211,7.390,148.295
C08440=1213.487,330.778,-71.464,-176.208,7.394,148.296
C08441=1213.482,331.026,-71.494,-176.206,7.396,148.296
C08442=1213.478,331.274,-71.526,-176.204,7.399,148.296
C08443=1213.474,331.522,-71.557,-176.202,7.402,148.296
C08444=1213.469,331.771,-71.589,-176.200,7.405,148.296
C08445=1213.465,332.019,-71.620,-176.198,7.407,148.296
C08446=1213.461,332.267,-71.652,-176.195,7.410,148.296
C08447=1213.456,332.515,-71.683,-176.194,7.413,148.296
C08448=1213.453,332.763,-71.715,-176.191,7.416,148.296
C08449=1213.448,333.010,-71.746,-176.190,7.419,148.296
C08450=1213.444,333.259,-71.777,-176.187,7.422,148.296
C08451=1213.440,333.506,-71.809,-176.185,7.424,148.297
C08452=1213.436,333.755,-71.840,-176.183,7.427,148.297
C08453=1213.431,334.002,-71.872,-176.181,7.430,148.297
C08454=1213.427,334.250,-71.904,-176.179,7.433,148.297
C08455=1213.423,334.498,-71.935,-176.177,7.435,148.297
C08456=1213.419,334.746,-71.966,-176.174,7.439,148.297
C08457=1213.415,334.994,-71.998,-176.173,7.441,148.297
C08458=1213.411,335.242,-72.030,-176.170,7.444,148.297
C08459=1213.406,335.491,-72.061,-176.168,7.448,148.298
C08460=1213.402,335.738,-72.093,-176.166,7.450,148.298
C08461=1213.398,335.986,-72.125,-176.164,7.453,148.298
C08462=1213.394,336.234,-72.156,-176.162,7.456,148.298
C08463=1213.390,336.482,-72.187,-176.160,7.459,148.298
C08464=1213.385,336.730,-72.219,-176.158,7.461,148.298
C08465=1213.381,336.978,-72.251,-176.155,7.465,148.298
C08466=1213.377,337.226,-72.283,-176.154,7.467,148.299
C08467=1213.373,337.474,-72.314,-176.151,7.470,148.299
C08468=1213.368,337.722,-72.346,-176.149,7.473,148.299
C08469=1213.364,337.969,-72.378,-176.147,7.476,148.299
C08470=1213.360,338.217,-72.410,-176.146,7.478,148.299
C08471=1213.357,338.465,-72.442,-176.143,7.482,148.299
C08472=1213.352,338.713,-72.474,-176.141,7.484,148.299
C08473=1213.348,338.961,-72.505,-176.139,7.487,148.300
C08474=1213.343,339.209,-72.536,-176.137,7.490,148.300
C08475=1213.340,339.457,-72.568,-176.135,7.493,148.300
C08476=1213.335,339.705,-72.601,-176.133,7.495,148.300
C08477=1213.331,339.953,-72.632,-176.131,7.499,148.300
C08478=1213.327,340.201,-72.664,-176.129,7.501,148.300
C08479=1213.323,340.449,-72.696,-176.127,7.505,148.301
C08480=1213.318,340.727,-72.732,-176.124,7.508,148.301
C08481=1213.313,341.005,-72.767,-176.122,7.511,148.301
C08482=1213.309,341.283,-72.803,-176.120,7.514,148.301
C08483=1213.304,341.561,-72.839,-176.118,7.517,148.301
C08484=1213.300,341.809,-72.871,-176.116,7.520,148.301
C08485=1213.295,342.057,-72.903,-176.114,7.523,148.301
C08486=1213.291,342.304,-72.935,-176.112,7.526,148.302
C08487=1213.287,342.553,-72.967,-176.110,7.528,148.302
C08488=1213.283,342.801,-72.999,-176.108,7.532,148.302
C08489=1213.279,343.048,-73.031,-176.106,7.534,148.302
C08490=1213.274,343.296,-73.063,-176.104,7.538,148.302
C08491=1213.271,343.544,-73.095,-176.102,7.540,148.303
C08492=1213.266,343.793,-73.127,-176.100,7.543,148.303
C08493=1213.262,344.040,-73.159,-176.098,7.546,148.303
C08494=1213.258,344.288,-73.192,-176.096,7.549,148.303
C08495=1213.254,344.536,-73.224,-176.094,7.552,148.303
C08496=1213.250,344.783,-73.255,-176.092,7.555,148.303
C08497=1213.245,345.032,-73.288,-176.090,7.557,148.304
C08498=1213.242,345.280,-73.320,-176.088,7.561,148.304
C08499=1213.236,345.527,-73.352,-176.087,7.563,148.304
C08500=1213.233,345.775,-73.384,-176.084,7.567,148.304
C08501=1213.229,346.023,-73.417,-176.083,7.569,148.304
C08502=1213.225,346.271,-73.449,-176.081,7.572,148.305
C08503=1213.220,346.519,-73.481,-176.079,7.575,148.305
C08504=1213.216,346.767,-73.513,-176.077,7.578,148.305
C08505=1213.212,347.014,-73.546,-176.075,7.581,148.305
C08506=1213.208,347.263,-73.578,-176.073,7.584,148.305
C08507=1213.203,347.510,-73.610,-176.071,7.587,148.306
C08508=1213.199,347.759,-73.642,-176.069,7.590,148.306
C08509=1213.195,348.006,-73.675,-176.067,7.593,148.306
C08510=1213.191,348.254,-73.707,-176.065,7.596,148.306
C08511=1213.187,348.502,-73.739,-176.064,7.598,148.306
C08512=1213.183,348.749,-73.772,-176.061,7.602,148.307
C08513=1213.178,348.998,-73.804,-176.060,7.604,148.307
C08514=1213.174,349.246,-73.836,-176.058,7.607,148.307
C08515=1213.170,349.493,-73.869,-176.056,7.610,148.307
C08516=1213.167,349.741,-73.901,-176.054,7.613,148.307
C08517=1213.162,349.989,-73.933,-176.052,7.616,148.308
C08518=1213.157,350.237,-73.966,-176.050,7.619,148.308
C08519=1213.154,350.485,-73.998,-176.048,7.622,148.308
C08520=1213.150,350.733,-74.031,-176.046,7.624,148.308
C08521=1213.146,350.981,-74.063,-176.044,7.628,148.308
C08522=1213.141,351.228,-74.096,-176.043,7.631,148.309
C08523=1213.137,351.476,-74.128,-176.041,7.634,148.309
C08524=1213.133,351.724,-74.160,-176.039,7.637,148.309
C08525=1213.129,351.972,-74.193,-176.037,7.640,148.310
C08526=1213.124,352.220,-74.226,-176.035,7.642,148.310
C08527=1213.121,352.468,-74.258,-176.034,7.645,148.310
C08528=1213.116,352.715,-74.290,-176.032,7.649,148.310
C08529=1213.112,352.963,-74.324,-176.030,7.651,148.310
C08530=1213.107,353.211,-74.356,-176.028,7.654,148.311
C08531=1213.104,353.459,-74.389,-176.026,7.657,148.311
C08532=1213.099,353.707,-74.421,-176.024,7.660,148.311
C08533=1213.095,353.955,-74.454,-176.023,7.663,148.311
C08534=1213.092,354.202,-74.487,-176.021,7.666,148.312
C08535=1213.087,354.451,-74.519,-176.019,7.669,148.312
C08536=1213.083,354.698,-74.552,-176.018,7.671,148.312
C08537=1213.078,354.946,-74.584,-176.015,7.675,148.312
C08538=1213.075,355.193,-74.617,-176.014,7.678,148.313
C08539=1213.071,355.441,-74.650,-176.012,7.681,148.313
C08540=1213.066,355.689,-74.682,-176.010,7.684,148.313
C08541=1213.062,355.937,-74.716,-176.008,7.687,148.313
C08542=1213.059,356.185,-74.748,-176.007,7.690,148.314
C08543=1213.054,356.433,-74.781,-176.005,7.692,148.314
C08544=1213.050,356.681,-74.814,-176.003,7.696,148.314
C08545=1213.046,356.928,-74.847,-176.002,7.698,148.315
C08546=1213.042,357.177,-74.879,-176.000,7.702,148.315
C08547=1213.038,357.423,-74.912,-175.998,7.704,148.315
C08548=1213.033,357.671,-74.945,-175.997,7.707,148.315
C08549=1213.029,357.920,-74.977,-175.995,7.710,148.316
C08550=1213.025,358.167,-75.010,-175.993,7.713,148.316
C08551=1213.021,358.415,-75.044,-175.991,7.717,148.316
C08552=1213.017,358.663,-75.077,-175.990,7.719,148.316
C08553=1213.013,358.911,-75.109,-175.988,7.723,148.317
C08554=1213.009,359.159,-75.142,-175.986,7.725,148.317
C08555=1213.005,359.406,-75.175,-175.985,7.728,148.317
C08556=1213.001,359.654,-75.208,-175.983,7.731,148.318
C08557=1212.996,359.902,-75.241,-175.981,7.734,148.318
C08558=1212.992,360.150,-75.274,-175.980,7.737,148.318
C08559=1212.988,360.398,-75.307,-175.978,7.740,148.318
C08560=1212.984,360.646,-75.340,-175.977,7.743,148.319
C08561=1212.980,360.893,-75.372,-175.974,7.746,148.319
C08562=1212.976,361.141,-75.406,-175.973,7.749,148.319
C08563=1212.972,361.388,-75.439,-175.972,7.752,148.320
C08564=1212.968,361.636,-75.472,-175.969,7.755,148.320
C08565=1212.964,361.884,-75.505,-175.968,7.758,148.320
C08566=1212.959,362.132,-75.538,-175.967,7.760,148.320
C08567=1212.955,362.380,-75.571,-175.965,7.764,148.321
C08568=1212.951,362.628,-75.604,-175.964,7.767,148.321
C08569=1212.947,362.875,-75.637,-175.962,7.769,148.321
C08570=1212.943,363.123,-75.670,-175.960,7.773,148.322
C08571=1212.939,363.371,-75.703,-175.959,7.775,148.322
C08572=1212.934,363.619,-75.736,-175.957,7.778,148.323
C08573=1212.930,363.866,-75.770,-175.955,7.782,148.323
C08574=1212.926,364.114,-75.803,-175.954,7.784,148.323
C08575=1212.922,364.362,-75.836,-175.953,7.787,148.324
C08576=1212.918,364.609,-75.869,-175.951,7.791,148.324
C08577=1212.914,364.857,-75.902,-175.949,7.793,148.324
C08578=1212.910,365.105,-75.935,-175.948,7.796,148.324
C08579=1212.905,365.353,-75.969,-175.946,7.800,148.325
C08580=1212.902,365.601,-76.002,-175.945,7.802,148.325
C08581=1212.898,365.849,-76.035,-175.943,7.805,148.325
C08582=1212.894,366.097,-76.068,-175.942,7.808,148.326
C08583=1212.890,366.344,-76.102,-175.940,7.811,148.326
C08584=1212.885,366.624,-76.139,-175.939,7.814,148.327
C08585=1212.881,366.904,-76.177,-175.937,7.818,148.327
C08586=1212.876,367.184,-76.215,-175.935,7.821,148.327
C08587=1212.871,367.465,-76.252,-175.933,7.825,148.328
C08588=1212.867,367.713,-76.285,-175.932,7.828,148.328
C08589=1212.863,367.960,-76.319,-175.931,7.830,148.329
C08590=1212.859,368.208,-76.352,-175.929,7.833,148.329
C08591=1212.855,368.455,-76.386,-175.928,7.837,148.329
C08592=1212.850,368.703,-76.419,-175.926,7.839,148.330
C08593=1212.846,368.951,-76.453,-175.925,7.842,148.330
C08594=1212.842,369.199,-76.486,-175.924,7.845,148.330
C08595=1212.838,369.446,-76.520,-175.922,7.848,148.331
C08596=1212.834,369.694,-76.553,-175.921,7.851,148.331
C08597=1212.830,369.942,-76.586,-175.919,7.854,148.331
C08598=1212.826,370.190,-76.619,-175.918,7.857,148.332
C08599=1212.822,370.437,-76.654,-175.917,7.860,148.332
C08600=1212.818,370.685,-76.687,-175.915,7.862,148.332
C08601=1212.813,370.933,-76.720,-175.914,7.866,148.333
C08602=1212.809,371.180,-76.753,-175.912,7.869,148.333
C08603=1212.805,371.427,-76.787,-175.911,7.871,148.334
C08604=1212.801,371.675,-76.820,-175.910,7.874,148.334
C08605=1212.797,371.924,-76.854,-175.909,7.877,148.334
C08606=1212.793,372.171,-76.888,-175.908,7.880,148.335
C08607=1212.789,372.419,-76.921,-175.906,7.883,148.335
C08608=1212.785,372.667,-76.955,-175.905,7.886,148.336
C08609=1212.781,372.914,-76.988,-175.903,7.889,148.336
C08610=1212.776,373.162,-77.022,-175.902,7.892,148.336
C08611=1212.773,373.410,-77.056,-175.901,7.895,148.337
C08612=1212.769,373.657,-77.090,-175.900,7.898,148.337
C08613=1212.765,373.905,-77.123,-175.899,7.900,148.338
C08614=1212.760,374.153,-77.157,-175.897,7.903,148.338
C08615=1212.756,374.400,-77.190,-175.896,7.906,148.338
C08616=1212.752,374.649,-77.224,-175.895,7.909,148.339
C08617=1212.749,374.896,-77.258,-175.894,7.912,148.339
C08618=1212.744,375.144,-77.292,-175.892,7.915,148.340
C08619=1212.740,375.391,-77.325,-175.891,7.918,148.340
C08620=1212.736,375.639,-77.359,-175.890,7.921,148.340
C08621=1212.732,375.887,-77.392,-175.889,7.924,148.341
C08622=1212.728,376.134,-77.427,-175.887,7.927,148.341
C08623=1212.724,376.382,-77.460,-175.886,7.929,148.341
C08624=1212.720,376.629,-77.494,-175.885,7.932,148.342
C08625=1212.715,376.877,-77.527,-175.884,7.935,148.342
C08626=1212.712,377.125,-77.562,-175.883,7.938,148.343
C08627=1212.707,377.373,-77.595,-175.882,7.941,148.343
C08628=1212.703,377.620,-77.629,-175.881,7.944,148.344
C08629=1212.699,377.868,-77.662,-175.879,7.947,148.344
C08630=1212.695,378.116,-77.697,-175.878,7.949,148.344
C08631=1212.691,378.363,-77.730,-175.877,7.952,148.345
C08632=1212.687,378.611,-77.764,-175.876,7.955,148.345
C08633=1212.683,378.859,-77.797,-175.875,7.958,148.346
C08634=1212.678,379.106,-77.832,-175.874,7.961,148.346
C08635=1212.675,379.354,-77.865,-175.873,7.964,148.347
C08636=1212.671,379.602,-77.899,-175.872,7.967,148.347
C08637=1212.666,379.849,-77.934,-175.870,7.969,148.347
C08638=1212.662,380.097,-77.967,-175.870,7.971,148.348
C08639=1212.659,380.345,-78.001,-175.869,7.974,148.348
C08640=1212.654,380.593,-78.035,-175.868,7.977,148.349
C08641=1212.650,380.840,-78.069,-175.867,7.980,148.349
C08642=1212.646,381.088,-78.104,-175.865,7.983,148.350
C08643=1212.642,381.336,-78.137,-175.865,7.986,148.350
C08644=1212.638,381.583,-78.171,-175.863,7.989,148.351
C08645=1212.634,381.830,-78.205,-175.862,7.992,148.351
C08646=1212.630,382.079,-78.239,-175.861,7.994,148.351
C08647=1212.625,382.326,-78.273,-175.860,7.998,148.352
C08648=1212.622,382.573,-78.307,-175.860,8.000,148.352
C08649=1212.617,382.821,-78.341,-175.858,8.002,148.353
C08650=1212.614,383.069,-78.375,-175.858,8.005,148.353
C08651=1212.610,383.316,-78.409,-175.856,8.008,148.354
C08652=1212.605,383.564,-78.443,-175.855,8.011,148.354
C08653=1212.602,383.812,-78.477,-175.855,8.014,148.355
C08654=1212.597,384.059,-78.511,-175.854,8.016,148.355
C08655=1212.593,384.307,-78.544,-175.853,8.019,148.355
C08656=1212.589,384.555,-78.579,-175.852,8.022,148.356
C08657=1212.585,384.802,-78.613,-175.851,8.025,148.356
C08658=1212.580,385.050,-78.648,-175.850,8.028,148.357
C08659=1212.577,385.298,-78.681,-175.849,8.030,148.357
C08660=1212.572,385.545,-78.716,-175.848,8.033,148.358
C08661=1212.569,385.793,-78.749,-175.847,8.036,148.358
C08662=1212.565,386.041,-78.784,-175.846,8.039,148.359
C08663=1212.561,386.288,-78.818,-175.846,8.041,148.359
C08664=1212.556,386.536,-78.852,-175.845,8.044,148.360
C08665=1212.553,386.784,-78.886,-175.844,8.047,148.360
C08666=1212.548,387.031,-78.921,-175.843,8.050,148.361
C08667=1212.544,387.278,-78.954,-175.842,8.052,148.361
C08668=1212.540,387.526,-78.989,-175.841,8.055,148.361
C08669=1212.536,387.773,-79.023,-175.840,8.058,148.362
C08670=1212.532,388.021,-79.057,-175.840,8.060,148.362
C08671=1212.528,388.269,-79.091,-175.839,8.063,148.363
C08672=1212.524,388.517,-79.126,-175.838,8.066,148.363
C08673=1212.520,388.764,-79.159,-175.837,8.068,148.364
C08674=1212.516,389.012,-79.194,-175.836,8.071,148.364
C08675=1212.511,389.259,-79.229,-175.836,8.074,148.365
C08676=1212.508,389.506,-79.263,-175.835,8.076,148.365
C08677=1212.504,389.755,-79.297,-175.834,8.079,148.366
C08678=1212.499,390.002,-79.331,-175.833,8.082,148.366
C08679=1212.495,390.250,-79.365,-175.833,8.084,148.367
C08680=1212.492,390.498,-79.399,-175.832,8.087,148.367
C08681=1212.487,390.745,-79.434,-175.831,8.090,148.368
C08682=1212.483,390.993,-79.469,-175.830,8.092,148.368
C08683=1212.479,391.240,-79.503,-175.829,8.095,148.369
C08684=1212.475,391.488,-79.537,-175.829,8.097,148.369
C08685=1212.471,391.735,-79.571,-175.828,8.100,148.369
C08686=1212.467,391.983,-79.606,-175.827,8.102,148.370
C08687=1212.463,392.231,-79.641,-175.827,8.105,148.370
C08688=1212.458,392.513,-79.679,-175.825,8.108,148.371
C08689=1212.454,392.795,-79.718,-175.825,8.111,148.371
C08690=1212.449,393.077,-79.758,-175.824,8.114,148.372
C08691=1212.445,393.360,-79.797,-175.823,8.117,148.373
C08692=1212.441,393.607,-79.831,-175.822,8.119,148.373
C08693=1212.436,393.854,-79.865,-175.822,8.122,148.374
C08694=1212.432,394.103,-79.900,-175.821,8.124,148.374
C08695=1212.429,394.350,-79.934,-175.820,8.127,148.374
C08696=1212.425,394.598,-79.969,-175.820,8.129,148.375
C08697=1212.420,394.845,-80.003,-175.819,8.132,148.375
C08698=1212.417,395.093,-80.038,-175.819,8.135,148.376
C08699=1212.412,395.340,-80.072,-175.817,8.138,148.376
C08700=1212.408,395.588,-80.107,-175.817,8.140,148.377
C08701=1212.405,395.835,-80.141,-175.816,8.143,148.377
C08702=1212.400,396.082,-80.176,-175.816,8.145,148.378
C08703=1212.396,396.331,-80.211,-175.815,8.147,148.378
C08704=1212.392,396.578,-80.245,-175.814,8.150,148.379
C08705=1212.388,396.826,-80.279,-175.814,8.152,148.379
C08706=1212.384,397.073,-80.314,-175.813,8.155,148.380
C08707=1212.379,397.321,-80.348,-175.813,8.157,148.380
C08708=1212.376,397.568,-80.383,-175.812,8.160,148.381
C08709=1212.371,397.816,-80.417,-175.811,8.162,148.381
C08710=1212.367,398.064,-80.452,-175.811,8.165,148.382
C08711=1212.364,398.310,-80.487,-175.810,8.168,148.382
C08712=1212.360,398.559,-80.521,-175.810,8.170,148.383
C08713=1212.355,398.806,-80.556,-175.809,8.172,148.383
C08714=1212.351,399.054,-80.591,-175.808,8.175,148.384
C08715=1212.348,399.301,-80.625,-175.808,8.177,148.384
C08716=1212.344,399.549,-80.659,-175.807,8.180,148.384
C08717=1212.339,399.796,-80.695,-175.807,8.182,148.385
C08718=1212.335,400.044,-80.729,-175.806,8.184,148.385
C08719=1212.332,400.291,-80.763,-175.805,8.187,148.386
C08720=1212.327,400.539,-80.798,-175.805,8.190,148.386
C08721=1212.323,400.787,-80.833,-175.805,8.192,148.387
C08722=1212.319,401.034,-80.868,-175.804,8.195,148.387
C08723=1212.316,401.282,-80.902,-175.804,8.197,148.388
C08724=1212.311,401.529,-80.936,-175.803,8.199,148.388
C08725=1212.307,401.777,-80.971,-175.803,8.201,148.389
C08726=1212.302,402.024,-81.006,-175.802,8.204,148.389
C08727=1212.300,402.272,-81.041,-175.801,8.206,148.390
C08728=1212.295,402.519,-81.075,-175.801,8.209,148.390
C08729=1212.291,402.767,-81.110,-175.800,8.211,148.391
C08730=1212.286,403.015,-81.144,-175.800,8.214,148.391
C08731=1212.283,403.262,-81.180,-175.800,8.216,148.392
C08732=1212.279,403.509,-81.214,-175.799,8.218,148.392
C08733=1212.275,403.757,-81.249,-175.798,8.221,148.393
C08734=1212.270,404.005,-81.283,-175.797,8.223,148.393
C08735=1212.267,404.252,-81.319,-175.797,8.225,148.394
C08736=1212.262,404.500,-81.353,-175.797,8.227,148.394
C08737=1212.259,404.748,-81.387,-175.796,8.229,148.394
C08738=1212.255,404.994,-81.423,-175.796,8.233,148.395
C08739=1212.251,405.242,-81.457,-175.795,8.235,148.396
C08740=1212.246,405.490,-81.492,-175.795,8.237,148.396
C08741=1212.242,405.737,-81.527,-175.795,8.239,148.396
C08742=1212.238,405.985,-81.562,-175.794,8.241,148.397
C08743=1212.235,406.233,-81.596,-175.793,8.244,148.397
C08744=1212.231,406.480,-81.632,-175.793,8.246,148.398
C08745=1212.226,406.727,-81.666,-175.792,8.248,148.398
C08746=1212.222,406.976,-81.701,-175.792,8.251,148.399
C08747=1212.218,407.222,-81.736,-175.791,8.253,148.399
C08748=1212.214,407.471,-81.771,-175.791,8.255,148.400
C08749=1212.210,407.718,-81.805,-175.790,8.258,148.400
C08750=1212.207,407.965,-81.840,-175.790,8.260,148.401
C08751=1212.202,408.213,-81.875,-175.790,8.262,148.401
C08752=1212.198,408.461,-81.910,-175.789,8.265,148.402
C08753=1212.194,408.707,-81.945,-175.789,8.266,148.402
C08754=1212.190,408.956,-81.980,-175.789,8.269,148.403
C08755=1212.186,409.203,-82.015,-175.788,8.271,148.403
C08756=1212.182,409.451,-82.050,-175.787,8.274,148.403
C08757=1212.178,409.698,-82.084,-175.787,8.276,148.404
C08758=1212.174,409.945,-82.119,-175.786,8.278,148.404
C08759=1212.170,410.193,-82.154,-175.786,8.280,148.405
C08760=1212.166,410.440,-82.189,-175.786,8.283,148.405
C08761=1212.162,410.688,-82.224,-175.785,8.285,148.406
C08762=1212.158,410.936,-82.260,-175.785,8.287,148.406
C08763=1212.154,411.183,-82.294,-175.784,8.289,148.407
C08764=1212.150,411.431,-82.329,-175.784,8.291,148.407
C08765=1212.146,411.678,-82.364,-175.784,8.293,148.408
C08766=1212.142,411.926,-82.398,-175.783,8.295,148.408
C08767=1212.138,412.173,-82.433,-175.783,8.298,148.409
C08768=1212.134,412.421,-82.468,-175.782,8.300,148.409
C08769=1212.130,412.668,-82.504,-175.782,8.303,148.409
C08770=1212.126,412.916,-82.538,-175.781,8.305,148.410
C08771=1212.122,413.163,-82.574,-175.781,8.307,148.410
C08772=1212.118,413.411,-82.608,-175.781,8.309,148.411
C08773=1212.114,413.658,-82.644,-175.780,8.311,148.411
C08774=1212.109,413.906,-82.678,-175.780,8.313,148.412
C08775=1212.106,414.153,-82.714,-175.779,8.315,148.412
C08776=1212.102,414.401,-82.749,-175.779,8.318,148.413
C08777=1212.097,414.648,-82.784,-175.779,8.320,148.413
C08778=1212.094,414.896,-82.819,-175.778,8.322,148.413
C08779=1212.089,415.143,-82.854,-175.778,8.324,148.414
C08780=1212.086,415.387,-82.888,-175.777,8.326,148.414
C08781=1212.082,415.630,-82.923,-175.777,8.328,148.415
C08782=1212.078,415.874,-82.958,-175.776,8.330,148.415
C08783=1212.074,416.118,-82.991,-175.776,8.333,148.416
C08784=1212.070,416.361,-83.026,-175.775,8.335,148.416
C08785=1212.066,416.604,-83.061,-175.776,8.336,148.417
C08786=1212.064,416.848,-83.095,-175.775,8.338,148.417
C08787=1212.066,417.091,-83.129,-175.775,8.340,148.417
C08788=1211.643,417.091,-83.165,-175.778,8.351,148.421
C08789=1211.643,416.847,-83.131,-175.778,8.349,148.421
C08790=1211.644,416.602,-83.097,-175.779,8.347,148.420
C08791=1211.648,416.357,-83.062,-175.779,8.345,148.420
C08792=1211.652,416.113,-83.027,-175.779,8.343,148.419
C08793=1211.656,415.867,-82.992,-175.780,8.341,148.419
C08794=1211.660,415.622,-82.957,-175.780,8.339,148.419
C08795=1211.664,415.378,-82.923,-175.780,8.337,148.418
C08796=1211.668,415.132,-82.889,-175.781,8.335,148.418
C08797=1211.672,414.885,-82.853,-175.781,8.333,148.417
C08798=1211.676,414.638,-82.818,-175.781,8.330,148.417
C08799=1211.680,414.390,-82.783,-175.782,8.328,148.416
C08800=1211.683,414.142,-82.748,-175.782,8.326,148.416
C08801=1211.688,413.895,-82.713,-175.783,8.324,148.415
C08802=1211.692,413.648,-82.678,-175.783,8.322,148.415
C08803=1211.696,413.400,-82.643,-175.783,8.320,148.414
C08804=1211.700,413.153,-82.608,-175.784,8.318,148.414
C08805=1211.704,412.905,-82.573,-175.784,8.315,148.414
C08806=1211.708,412.658,-82.538,-175.785,8.313,148.413
C08807=1211.712,412.410,-82.503,-175.786,8.310,148.413
C08808=1211.716,412.163,-82.468,-175.786,8.308,148.412
C08809=1211.720,411.915,-82.433,-175.787,8.306,148.412
C08810=1211.725,411.667,-82.399,-175.787,8.304,148.411
C08811=1211.728,411.420,-82.364,-175.787,8.302,148.411
C08812=1211.732,411.172,-82.329,-175.788,8.299,148.410
C08813=1211.736,410.925,-82.294,-175.788,8.297,148.410
C08814=1211.740,410.677,-82.259,-175.789,8.295,148.409
C08815=1211.744,410.430,-82.224,-175.789,8.293,148.409
C08816=1211.748,410.182,-82.189,-175.789,8.291,148.408
C08817=1211.753,409.935,-82.154,-175.790,8.289,148.408
C08818=1211.757,409.687,-82.119,-175.790,8.286,148.408
C08819=1211.761,409.439,-82.084,-175.790,8.284,148.407
C08820=1211.765,409.192,-82.049,-175.791,8.281,148.407
C08821=1211.768,408.944,-82.014,-175.791,8.279,148.406
C08822=1211.772,408.698,-81.979,-175.792,8.277,148.406
C08823=1211.776,408.450,-81.944,-175.792,8.275,148.405
C08824=1211.781,408.202,-81.910,-175.793,8.273,148.405
C08825=1211.784,407.955,-81.874,-175.793,8.271,148.404
C08826=1211.789,407.707,-81.840,-175.793,8.268,148.404
C08827=1211.793,407.460,-81.804,-175.794,8.266,148.403
C08828=1211.797,407.212,-81.770,-175.795,8.263,148.403
C08829=1211.801,406.964,-81.736,-175.795,8.261,148.402
C08830=1211.804,406.717,-81.700,-175.796,8.259,148.402
C08831=1211.809,406.470,-81.666,-175.796,8.257,148.401
C08832=1211.813,406.221,-81.631,-175.796,8.254,148.401
C08833=1211.817,405.975,-81.596,-175.797,8.253,148.401
C08834=1211.821,405.727,-81.561,-175.797,8.249,148.400
C08835=1211.825,405.479,-81.527,-175.798,8.247,148.399
C08836=1211.828,405.232,-81.491,-175.798,8.245,148.399
C08837=1211.833,404.984,-81.457,-175.799,8.243,148.399
C08838=1211.837,404.736,-81.422,-175.799,8.241,148.398
C08839=1211.841,404.490,-81.387,-175.800,8.238,148.398
C08840=1211.845,404.241,-81.352,-175.800,8.236,148.397
C08841=1211.849,403.994,-81.318,-175.801,8.234,148.397
C08842=1211.853,403.747,-81.283,-175.801,8.231,148.396
C08843=1211.857,403.499,-81.248,-175.802,8.228,148.396
C08844=1211.861,403.251,-81.213,-175.802,8.226,148.395
C08845=1211.866,403.004,-81.179,-175.803,8.224,148.395
C08846=1211.869,402.757,-81.144,-175.803,8.222,148.394
C08847=1211.873,402.509,-81.109,-175.804,8.219,148.394
C08848=1211.877,402.261,-81.075,-175.804,8.217,148.393
C08849=1211.882,402.014,-81.040,-175.805,8.215,148.393
C08850=1211.885,401.766,-81.005,-175.805,8.212,148.392
C08851=1211.889,401.519,-80.971,-175.806,8.209,148.392
C08852=1211.893,401.271,-80.936,-175.807,8.207,148.391
C08853=1211.898,401.024,-80.901,-175.807,8.205,148.391
C08854=1211.902,400.776,-80.866,-175.807,8.202,148.390
C08855=1211.905,400.529,-80.832,-175.808,8.200,148.390
C08856=1211.909,400.281,-80.797,-175.808,8.198,148.389
C08857=1211.914,400.033,-80.763,-175.810,8.195,148.389
C08858=1211.918,399.785,-80.728,-175.810,8.193,148.389
C08859=1211.921,399.539,-80.693,-175.810,8.190,148.388
C08860=1211.925,399.291,-80.659,-175.811,8.187,148.388
C08861=1211.930,399.043,-80.624,-175.811,8.185,148.387
C08862=1211.934,398.795,-80.589,-175.812,8.183,148.387
C08863=1211.938,398.548,-80.555,-175.813,8.180,148.386
C08864=1211.942,398.300,-80.521,-175.813,8.178,148.386
C08865=1211.946,398.053,-80.485,-175.814,8.176,148.385
C08866=1211.950,397.805,-80.450,-175.814,8.173,148.385
C08867=1211.954,397.558,-80.417,-175.815,8.171,148.384
C08868=1211.958,397.310,-80.382,-175.816,8.168,148.384
C08869=1211.962,397.062,-80.347,-175.816,8.165,148.383
C08870=1211.966,396.815,-80.313,-175.817,8.163,148.383
C08871=1211.970,396.567,-80.279,-175.817,8.160,148.382
C08872=1211.975,396.320,-80.244,-175.818,8.158,148.382
C08873=1211.978,396.072,-80.210,-175.819,8.155,148.381
C08874=1211.982,395.825,-80.175,-175.819,8.153,148.381
C08875=1211.986,395.577,-80.140,-175.820,8.150,148.380
C08876=1211.991,395.330,-80.105,-175.820,8.148,148.380
C08877=1211.995,395.082,-80.072,-175.822,8.145,148.379
C08878=1211.999,394.834,-80.037,-175.822,8.143,148.379
C08879=1212.003,394.587,-80.002,-175.823,8.140,148.378
C08880=1212.006,394.339,-79.968,-175.823,8.138,148.378
C08881=1212.011,394.092,-79.934,-175.824,8.135,148.377
C08882=1212.014,393.844,-79.899,-175.825,8.133,148.377
C08883=1212.019,393.596,-79.865,-175.825,8.130,148.376
C08884=1212.023,393.349,-79.830,-175.826,8.128,148.376
C08885=1212.028,393.067,-79.791,-175.827,8.124,148.376
C08886=1212.032,392.785,-79.752,-175.828,8.121,148.375
C08887=1212.036,392.502,-79.713,-175.828,8.118,148.374
C08888=1212.041,392.220,-79.674,-175.830,8.115,148.374
C08889=1212.045,391.972,-79.639,-175.830,8.113,148.373
C08890=1212.049,391.725,-79.605,-175.830,8.110,148.373
C08891=1212.053,391.477,-79.570,-175.831,8.108,148.372
C08892=1212.058,391.229,-79.536,-175.832,8.105,148.372
C08893=1212.062,390.982,-79.502,-175.833,8.102,148.371
C08894=1212.066,390.734,-79.467,-175.833,8.100,148.371
C08895=1212.069,390.487,-79.433,-175.834,8.097,148.371
C08896=1212.073,390.239,-79.398,-175.835,8.095,148.370
C08897=1212.077,389.992,-79.365,-175.836,8.092,148.370
C08898=1212.082,389.744,-79.330,-175.837,8.089,148.369
C08899=1212.086,389.496,-79.295,-175.837,8.087,148.369
C08900=1212.090,389.249,-79.261,-175.838,8.084,148.368
C08901=1212.094,389.001,-79.228,-175.839,8.081,148.368
C08902=1212.098,388.753,-79.193,-175.839,8.079,148.367
C08903=1212.102,388.506,-79.159,-175.841,8.076,148.367
C08904=1212.106,388.259,-79.125,-175.841,8.073,148.366
C08905=1212.110,388.011,-79.090,-175.842,8.071,148.366
C08906=1212.115,387.763,-79.056,-175.843,8.068,148.365
C08907=1212.118,387.515,-79.022,-175.844,8.065,148.365
C08908=1212.122,387.268,-78.987,-175.845,8.062,148.364
C08909=1212.127,387.020,-78.954,-175.845,8.060,148.364
C08910=1212.131,386.772,-78.919,-175.847,8.057,148.364
C08911=1212.134,386.525,-78.885,-175.847,8.054,148.363
C08912=1212.139,386.278,-78.851,-175.848,8.052,148.363
C08913=1212.142,386.030,-78.817,-175.849,8.049,148.362
C08914=1212.147,385.782,-78.783,-175.850,8.046,148.362
C08915=1212.151,385.535,-78.749,-175.851,8.043,148.361
C08916=1212.155,385.287,-78.714,-175.852,8.040,148.361
C08917=1212.159,385.039,-78.680,-175.853,8.038,148.360
C08918=1212.163,384.792,-78.646,-175.854,8.035,148.360
C08919=1212.167,384.544,-78.612,-175.854,8.032,148.359
C08920=1212.171,384.296,-78.578,-175.856,8.029,148.359
C08921=1212.175,384.049,-78.544,-175.856,8.027,148.358
C08922=1212.179,383.801,-78.509,-175.857,8.024,148.358
C08923=1212.183,383.553,-78.476,-175.858,8.021,148.358
C08924=1212.187,383.306,-78.442,-175.859,8.018,148.357
C08925=1212.192,383.059,-78.408,-175.860,8.016,148.357
C08926=1212.195,382.810,-78.374,-175.861,8.013,148.356
C08927=1212.200,382.563,-78.340,-175.863,8.010,148.356
C08928=1212.204,382.316,-78.306,-175.863,8.008,148.355
C08929=1212.208,382.067,-78.272,-175.864,8.005,148.355
C08930=1212.212,381.820,-78.238,-175.865,8.002,148.354
C08931=1212.216,381.572,-78.203,-175.866,7.999,148.354
C08932=1212.220,381.325,-78.170,-175.867,7.996,148.353
C08933=1212.224,381.077,-78.136,-175.868,7.993,148.353
C08934=1212.228,380.829,-78.101,-175.870,7.990,148.353
C08935=1212.232,380.582,-78.068,-175.870,7.987,148.352
C08936=1212.236,380.334,-78.033,-175.871,7.985,148.352
C08937=1212.240,380.087,-78.000,-175.872,7.983,148.351
C08938=1212.244,379.839,-77.966,-175.873,7.980,148.351
C08939=1212.249,379.591,-77.932,-175.874,7.977,148.350
C08940=1212.252,379.343,-77.898,-175.875,7.974,148.350
C08941=1212.256,379.096,-77.865,-175.876,7.971,148.350
C08942=1212.261,378.848,-77.830,-175.878,7.968,148.349
C08943=1212.265,378.601,-77.797,-175.879,7.965,148.349
C08944=1212.269,378.353,-77.762,-175.880,7.962,148.348
C08945=1212.273,378.105,-77.729,-175.881,7.959,148.348
C08946=1212.277,377.858,-77.695,-175.882,7.957,148.347
C08947=1212.282,377.610,-77.661,-175.883,7.954,148.347
C08948=1212.286,377.363,-77.627,-175.884,7.951,148.347
C08949=1212.289,377.114,-77.594,-175.886,7.948,148.346
C08950=1212.294,376.867,-77.559,-175.887,7.945,148.346
C08951=1212.298,376.619,-77.526,-175.888,7.942,148.345
C08952=1212.302,376.372,-77.492,-175.889,7.939,148.345
C08953=1212.305,376.123,-77.459,-175.890,7.937,148.344
C08954=1212.310,375.876,-77.424,-175.891,7.934,148.344
C08955=1212.314,375.628,-77.391,-175.892,7.931,148.344
C08956=1212.318,375.381,-77.357,-175.894,7.928,148.343
C08957=1212.323,375.133,-77.324,-175.895,7.925,148.343
C08958=1212.326,374.885,-77.290,-175.896,7.922,148.342
C08959=1212.330,374.638,-77.256,-175.898,7.919,148.342
C08960=1212.334,374.390,-77.223,-175.899,7.916,148.342
C08961=1212.339,374.142,-77.189,-175.900,7.913,148.341
C08962=1212.343,373.895,-77.155,-175.901,7.911,148.341
C08963=1212.346,373.646,-77.122,-175.902,7.908,148.340
C08964=1212.350,373.399,-77.088,-175.904,7.905,148.340
C08965=1212.355,373.151,-77.054,-175.905,7.902,148.340
C08966=1212.359,372.904,-77.020,-175.906,7.899,148.339
C08967=1212.363,372.656,-76.987,-175.907,7.896,148.339
C08968=1212.367,372.409,-76.954,-175.909,7.893,148.338
C08969=1212.370,372.161,-76.920,-175.910,7.890,148.338
C08970=1212.375,371.913,-76.886,-175.911,7.887,148.338
C08971=1212.379,371.665,-76.853,-175.913,7.884,148.337
C08972=1212.384,371.417,-76.820,-175.914,7.882,148.337
C08973=1212.387,371.170,-76.786,-175.915,7.879,148.337
C08974=1212.392,370.922,-76.753,-175.917,7.875,148.336
C08975=1212.396,370.674,-76.719,-175.918,7.873,148.336
C08976=1212.400,370.427,-76.685,-175.920,7.870,148.335
C08977=1212.404,370.179,-76.652,-175.921,7.867,148.335
C08978=1212.408,369.931,-76.618,-175.922,7.864,148.335
C08979=1212.412,369.683,-76.585,-175.924,7.860,148.334
C08980=1212.416,369.436,-76.551,-175.925,7.858,148.334
C08981=1212.420,369.189,-76.518,-175.926,7.855,148.333
C08982=1212.425,368.941,-76.485,-175.928,7.852,148.333
C08983=1212.429,368.693,-76.451,-175.929,7.850,148.333
C08984=1212.433,368.444,-76.418,-175.931,7.846,148.332
C08985=1212.436,368.197,-76.384,-175.932,7.843,148.332
C08986=1212.441,367.950,-76.351,-175.934,7.841,148.332
C08987=1212.445,367.702,-76.318,-175.935,7.838,148.331
C08988=1212.449,367.454,-76.285,-175.936,7.834,148.331
C08989=1212.454,367.174,-76.246,-175.938,7.831,148.331
C08990=1212.459,366.893,-76.209,-175.939,7.828,148.330
C08991=1212.463,366.614,-76.172,-175.942,7.824,148.330
C08992=1212.467,366.333,-76.134,-175.943,7.821,148.330
C08993=1212.471,366.086,-76.101,-175.945,7.818,148.329
C08994=1212.475,365.838,-76.068,-175.946,7.815,148.329
C08995=1212.480,365.590,-76.034,-175.947,7.812,148.329
C08996=1212.484,365.342,-76.001,-175.949,7.809,148.328
C08997=1212.489,365.094,-75.967,-175.950,7.806,148.328
C08998=1212.493,364.847,-75.934,-175.952,7.803,148.328
C08999=1212.497,364.599,-75.901,-175.954,7.800,148.327
C09000=1212.501,364.351,-75.868,-175.955,7.797,148.327
C09001=1212.505,364.104,-75.835,-175.957,7.795,148.327
C09002=1212.509,363.856,-75.802,-175.958,7.791,148.326
C09003=1212.513,363.607,-75.768,-175.960,7.788,148.326
C09004=1212.517,363.360,-75.735,-175.961,7.786,148.325
C09005=1212.521,363.112,-75.702,-175.963,7.782,148.325
C09006=1212.525,362.864,-75.669,-175.965,7.779,148.325
C09007=1212.529,362.617,-75.636,-175.966,7.777,148.324
C09008=1212.533,362.369,-75.603,-175.968,7.773,148.324
C09009=1212.537,362.121,-75.570,-175.969,7.770,148.324
C09010=1212.541,361.874,-75.537,-175.971,7.768,148.324
C09011=1212.545,361.626,-75.503,-175.973,7.764,148.323
C09012=1212.549,361.378,-75.470,-175.974,7.762,148.323
C09013=1212.553,361.130,-75.437,-175.975,7.759,148.323
C09014=1212.558,360.883,-75.404,-175.978,7.756,148.322
C09015=1212.562,360.634,-75.372,-175.979,7.753,148.322
C09016=1212.566,360.387,-75.338,-175.981,7.749,148.322
C09017=1212.570,360.139,-75.305,-175.983,7.747,148.322
C09018=1212.574,359.891,-75.272,-175.984,7.744,148.321
C09019=1212.578,359.644,-75.240,-175.986,7.741,148.321
C09020=1212.582,359.396,-75.206,-175.987,7.738,148.321
C09021=1212.586,359.148,-75.174,-175.989,7.735,148.320
C09022=1212.591,358.900,-75.141,-175.991,7.732,148.320
C09023=1212.595,358.652,-75.108,-175.992,7.729,148.320
C09024=1212.599,358.405,-75.075,-175.994,7.726,148.320
C09025=1212.604,358.157,-75.042,-175.996,7.723,148.319
C09026=1212.607,357.909,-75.010,-175.998,7.720,148.319
C09027=1212.611,357.662,-74.977,-175.999,7.717,148.319
C09028=1212.616,357.414,-74.944,-176.001,7.714,148.318
C09029=1212.620,357.166,-74.911,-176.003,7.711,148.318
C09030=1212.624,356.918,-74.878,-176.005,7.708,148.318
C09031=1212.628,356.670,-74.845,-176.006,7.705,148.317
C09032=1212.632,356.423,-74.812,-176.008,7.702,148.317
C09033=1212.636,356.174,-74.780,-176.010,7.699,148.317
C09034=1212.640,355.927,-74.747,-176.011,7.696,148.317
C09035=1212.645,355.678,-74.714,-176.013,7.694,148.317
C09036=1212.649,355.430,-74.681,-176.015,7.690,148.316
C09037=1212.652,355.183,-74.648,-176.017,7.688,148.316
C09038=1212.657,354.935,-74.616,-176.019,7.684,148.316
C09039=1212.661,354.688,-74.583,-176.020,7.682,148.315
C09040=1212.666,354.440,-74.550,-176.022,7.678,148.315
C09041=1212.669,354.192,-74.518,-176.024,7.676,148.315
C09042=1212.673,353.944,-74.485,-176.026,7.672,148.315
C09043=1212.678,353.696,-74.453,-176.027,7.670,148.314
C09044=1212.681,353.448,-74.420,-176.029,7.667,148.314
C09045=1212.686,353.200,-74.388,-176.031,7.664,148.314
C09046=1212.690,352.953,-74.355,-176.033,7.661,148.314
C09047=1212.695,352.705,-74.322,-176.035,7.658,148.313
C09048=1212.698,352.457,-74.290,-176.036,7.655,148.313
C09049=1212.703,352.209,-74.257,-176.039,7.652,148.313
C09050=1212.707,351.961,-74.224,-176.040,7.649,148.313
C09051=1212.711,351.713,-74.192,-176.042,7.646,148.313
C09052=1212.715,351.465,-74.159,-176.044,7.643,148.312
C09053=1212.720,351.218,-74.127,-176.046,7.640,148.312
C09054=1212.723,350.970,-74.095,-176.047,7.637,148.312
C09055=1212.728,350.722,-74.062,-176.049,7.635,148.312
C09056=1212.732,350.474,-74.029,-176.051,7.631,148.311
C09057=1212.735,350.226,-73.997,-176.053,7.629,148.311
C09058=1212.740,349.979,-73.965,-176.055,7.625,148.311
C09059=1212.744,349.731,-73.933,-176.057,7.623,148.311
C09060=1212.748,349.483,-73.900,-176.059,7.619,148.311
C09061=1212.752,349.235,-73.867,-176.061,7.617,148.310
C09062=1212.756,348.987,-73.835,-176.063,7.614,148.310
C09063=1212.761,348.739,-73.803,-176.065,7.611,148.310
C09064=1212.765,348.492,-73.770,-176.067,7.608,148.310
C09065=1212.769,348.244,-73.738,-176.068,7.605,148.309
C09066=1212.773,347.995,-73.706,-176.070,7.602,148.309
C09067=1212.777,347.748,-73.673,-176.072,7.599,148.309
C09068=1212.782,347.500,-73.641,-176.074,7.596,148.309
C09069=1212.786,347.252,-73.609,-176.076,7.593,148.309
C09070=1212.790,347.004,-73.577,-176.078,7.590,148.308
C09071=1212.793,346.756,-73.544,-176.079,7.587,148.308
C09072=1212.799,346.509,-73.512,-176.082,7.584,148.308
C09073=1212.802,346.261,-73.480,-176.083,7.581,148.308
C09074=1212.807,346.012,-73.448,-176.086,7.578,148.308
C09075=1212.810,345.765,-73.415,-176.088,7.576,148.308
C09076=1212.815,345.517,-73.383,-176.090,7.573,148.307
C09077=1212.819,345.269,-73.351,-176.091,7.570,148.307
C09078=1212.823,345.021,-73.319,-176.093,7.568,148.307
C09079=1212.827,344.773,-73.287,-176.095,7.564,148.307
C09080=1212.832,344.525,-73.255,-176.097,7.562,148.307
C09081=1212.835,344.278,-73.222,-176.099,7.558,148.306
C09082=1212.840,344.029,-73.190,-176.101,7.556,148.306
C09083=1212.844,343.782,-73.158,-176.103,7.552,148.306
C09084=1212.849,343.534,-73.126,-176.105,7.550,148.306
C09085=1212.852,343.286,-73.094,-176.107,7.547,148.306
C09086=1212.857,343.038,-73.062,-176.109,7.544,148.306
C09087=1212.861,342.790,-73.030,-176.111,7.541,148.305
C09088=1212.865,342.542,-72.998,-176.113,7.539,148.305
C09089=1212.869,342.294,-72.966,-176.115,7.535,148.305
C09090=1212.874,342.046,-72.934,-176.117,7.533,148.305
C09091=1212.878,341.798,-72.902,-176.119,7.529,148.305
C09092=1212.882,341.550,-72.870,-176.121,7.526,148.304
C09093=1212.887,341.272,-72.834,-176.123,7.524,148.304
C09094=1212.891,340.995,-72.798,-176.125,7.520,148.304
C09095=1212.896,340.716,-72.763,-176.128,7.517,148.304
C09096=1212.901,340.439,-72.727,-176.130,7.514,148.304
C09097=1212.905,340.190,-72.695,-176.132,7.510,148.303
C09098=1212.909,339.942,-72.663,-176.134,7.508,148.303
C09099=1212.913,339.695,-72.632,-176.136,7.505,148.303
C09100=1212.917,339.447,-72.600,-176.138,7.502,148.303
C09101=1212.921,339.198,-72.567,-176.140,7.499,148.303
C09102=1212.926,338.951,-72.536,-176.142,7.497,148.303
C09103=1212.929,338.703,-72.504,-176.144,7.493,148.303
C09104=1212.934,338.455,-72.472,-176.146,7.491,148.302
C09105=1212.938,338.207,-72.441,-176.148,7.487,148.302
C09106=1212.942,337.959,-72.409,-176.150,7.485,148.302
C09107=1212.946,337.711,-72.377,-176.153,7.482,148.302
C09108=1212.951,337.463,-72.345,-176.154,7.479,148.302
C09109=1212.955,337.216,-72.313,-176.157,7.476,148.302
C09110=1212.959,336.968,-72.282,-176.159,7.474,148.302
C09111=1212.963,336.719,-72.250,-176.161,7.470,148.302
C09112=1212.968,336.471,-72.218,-176.162,7.468,148.301
C09113=1212.972,336.223,-72.187,-176.165,7.465,148.301
C09114=1212.976,335.976,-72.155,-176.167,7.462,148.301
C09115=1212.980,335.727,-72.124,-176.169,7.459,148.301
C09116=1212.985,335.480,-72.092,-176.172,7.456,148.301
C09117=1212.989,335.232,-72.060,-176.173,7.453,148.301
C09118=1212.992,334.984,-72.028,-176.175,7.450,148.301
C09119=1212.997,334.736,-71.997,-176.178,7.448,148.301
C09120=1213.001,334.488,-71.966,-176.180,7.445,148.300
C09121=1213.005,334.240,-71.934,-176.181,7.442,148.300
C09122=1213.010,333.991,-71.902,-176.184,7.439,148.300
C09123=1213.014,333.744,-71.871,-176.186,7.436,148.300
C09124=1213.018,333.496,-71.839,-176.188,7.433,148.300
C09125=1213.022,333.248,-71.808,-176.190,7.431,148.300
C09126=1213.026,333.000,-71.776,-176.192,7.428,148.300
C09127=1213.031,332.752,-71.746,-176.194,7.425,148.300
C09128=1213.034,332.504,-71.714,-176.197,7.422,148.299
C09129=1213.039,332.257,-71.682,-176.199,7.420,148.299
C09130=1213.044,332.008,-71.651,-176.201,7.416,148.299
C09131=1213.048,331.760,-71.619,-176.203,7.414,148.299
